   cmAnodeMainPnP1AxisZ.commandConfiguration.gearInVelocity.positionControlled := FALSE;
   cmAnodeMainPnP1AxisZ.commandConfiguration.camIn.masterOffset := 0.0;
   cmAnodeMainPnP1AxisZ.commandConfiguration.camIn.slaveOffset := 0.0;
   cmAnodeMainPnP1AxisZ.commandConfiguration.camIn.masterScaling := 1.0;
   cmAnodeMainPnP1AxisZ.commandConfiguration.camIn.slaveScaling := 1.0;
   cmAnodeMainPnP1AxisZ.commandConfiguration.camIn.masterSyncPosition := 0.0;
   cmAnodeMainPnP1AxisZ.commandConfiguration.camIn.syncProfileReference := 1;
   cmAnodeMainPnP1AxisZ.commandConfiguration.camIn.masterStartDistance := 0.0;
   cmAnodeMainPnP1AxisZ.commandConfiguration.camIn.velocity := -1.0;
   cmAnodeMainPnP1AxisZ.commandConfiguration.camIn.acceleration := -1.0;
   cmAnodeMainPnP1AxisZ.commandConfiguration.camIn.deceleration := -1.0;
   cmAnodeMainPnP1AxisZ.commandConfiguration.camIn.jerk := -1.0;
   cmAnodeMainPnP1AxisZ.commandConfiguration.camIn.applicationMode := 0;
   cmAnodeMainPnP1AxisZ.commandConfiguration.camIn.syncDirection := 1;
   cmAnodeMainPnP1AxisZ.commandConfiguration.gearOutCamOut.slavePosition := 0.0;
   cmAnodeMainPnP1AxisZ.commandConfiguration.gearOutCamOut.syncProfileReference := 1;
   cmAnodeMainPnP1AxisZ.commandConfiguration.gearOutCamOut.masterStopDistance := 0.0;
   cmAnodeMainPnP1AxisZ.commandConfiguration.gearOutCamOut.deceleration := -1.0;
   cmAnodeMainPnP1AxisZ.commandConfiguration.gearOutCamOut.jerk := -1.0;
   cmAnodeMainPnP1AxisZ.commandConfiguration.gearOutCamOut.syncOutDirection := 3;
   cmAnodeMainPnP1AxisZ.commandConfiguration.gearOutCamOut.gearOutCamOutMode := -1;
   cmAnodeMainPnP1AxisZ.commandConfiguration.phasing.phaseShift := 0.0;
   cmAnodeMainPnP1AxisZ.commandConfiguration.phasing.velocity := -1.0;
   cmAnodeMainPnP1AxisZ.commandConfiguration.phasing.acceleration := -1.0;
   cmAnodeMainPnP1AxisZ.commandConfiguration.phasing.deceleration := -1.0;
   cmAnodeMainPnP1AxisZ.commandConfiguration.phasing.jerk := -1.0;
   cmAnodeMainPnP1AxisZ.commandConfiguration.phasing.profileReference := 0;
   cmAnodeMainPnP1AxisZ.commandConfiguration.phasing.phasingDistance := 0.0;
   cmAnodeMainPnP1AxisZ.commandConfiguration.phasing.startPosition := 0.0;
   cmAnodeMainPnP1AxisZ.commandConfiguration.phasing.direction := 3;
   cmAnodeMainPnP1AxisZ.commandConfiguration.phasing.phaseAbsolute := TRUE;
   cmAnodeMainPnP1AxisZ.commandConfiguration.phasing.phaseShiftChangeOnTheFly := FALSE;
   cmAnodeMainPnP1AxisZ.commandConfiguration.offset.offset := 0.0;
   cmAnodeMainPnP1AxisZ.commandConfiguration.offset.profileReference := 1;
   cmAnodeMainPnP1AxisZ.commandConfiguration.offset.offsetDistance := 0.0;
   cmAnodeMainPnP1AxisZ.commandConfiguration.offset.startPosition := 0.0;
   cmAnodeMainPnP1AxisZ.commandConfiguration.offset.direction := 3;
   cmAnodeMainPnP1AxisZ.commandConfiguration.offset.offsetAbsolute := TRUE;
   cmAnodeMainPnP1AxisZ.commandConfiguration.offset.offsetChangeOnTheFly := FALSE;
   cmAnodeMainPnP1AxisZ.commands.enableMasterControl := TRUE;
   cmAnodeMainPnP1AxisZ.commands.enableAxis := FALSE;
   cmAnodeMainPnP1AxisZ.commands.resetAxis := FALSE;
   cmAnodeMainPnP1AxisZ.commands.openBrake := FALSE;
   cmAnodeMainPnP1AxisZ.commands.jogForward := FALSE;
   cmAnodeMainPnP1AxisZ.commands.jogBackward := FALSE;
   cmAnodeMainPnP1AxisZ.commands.moveVelocity := FALSE;
   cmAnodeMainPnP1AxisZ.commands.stop := FALSE;
   cmAnodeMainPnP1AxisZ.commands.fastStop := FALSE;
   cmAnodeMainPnP1AxisZ.commands.torqueLimiting := FALSE;
   cmAnodeMainPnP1AxisZ.commands.homing := FALSE;
   cmAnodeMainPnP1AxisZ.commands.posRelative := FALSE;
   cmAnodeMainPnP1AxisZ.commands.posAbsolute := FALSE;
   cmAnodeMainPnP1AxisZ.commands.posSuperimposed := FALSE;
   cmAnodeMainPnP1AxisZ.commands.haltSuperimposed := FALSE;
   cmAnodeMainPnP1AxisZ.commands.selectSetPosition := 3;
   cmAnodeMainPnP1AxisZ.commands.uploadParameters := FALSE;
   cmAnodeMainPnP1AxisZ.commands.refreshConfiguration := FALSE;
   cmAnodeMainPnP1AxisZ.commands.editConfiguration := FALSE;
   cmAnodeMainPnP1AxisZ.commands.saveConfiguration := FALSE;
   cmAnodeMainPnP1AxisZ.commands.uploadCurrentTorque := FALSE;
   cmAnodeMainPnP1AxisZ.commands.reset := FALSE;
   cmAnodeMainPnP1AxisZ.monitoring.enable := TRUE;
   cmAnodeMainPnP1AxisZ.monitoring.referenceDesignator := WSTRING#'AnodeMainPnP1AxisZ';
   cmAnodeMainPnP1AxisZ.monitoring.enabled := TRUE;
   cmAnodeMainPnP1AxisZ.monitoring.enableManualCmds := FALSE;
   cmAnodeMainPnP1AxisZ.monitoring.reset := FALSE;
   cmAnodeMainPnP1AxisZ.monitoring.resetAxis := FALSE;
   cmAnodeMainPnP1AxisZ.monitoring.enableAxis := TRUE;
   cmAnodeMainPnP1AxisZ.monitoring.openBrake := FALSE;
   cmAnodeMainPnP1AxisZ.monitoring.jogBackward := FALSE;
   cmAnodeMainPnP1AxisZ.monitoring.jogForward := FALSE;
   cmAnodeMainPnP1AxisZ.monitoring.moveVelocity := FALSE;
   cmAnodeMainPnP1AxisZ.monitoring.stop := FALSE;
   cmAnodeMainPnP1AxisZ.monitoring.fastStop := FALSE;
   cmAnodeMainPnP1AxisZ.monitoring.torqueLimiting := FALSE;
   cmAnodeMainPnP1AxisZ.monitoring.homing := FALSE;
   cmAnodeMainPnP1AxisZ.monitoring.posRelative := FALSE;
   cmAnodeMainPnP1AxisZ.monitoring.posAbsolute := FALSE;
   cmAnodeMainPnP1AxisZ.monitoring.posSuperimposed := FALSE;
   cmAnodeMainPnP1AxisZ.monitoring.haltSuperimposed := FALSE;
   cmAnodeMainPnP1AxisZ.monitoring.brakeOpened := FALSE;
   cmAnodeMainPnP1AxisZ.monitoring.axisEnabled := TRUE;
   cmAnodeMainPnP1AxisZ.monitoring.resetActive := FALSE;
   cmAnodeMainPnP1AxisZ.monitoring.inVelocity := FALSE;
   cmAnodeMainPnP1AxisZ.monitoring.inLimitation := FALSE;
   cmAnodeMainPnP1AxisZ.monitoring.inClamping := FALSE;
   cmAnodeMainPnP1AxisZ.monitoring.startSync := FALSE;
   cmAnodeMainPnP1AxisZ.monitoring.inSync := FALSE;
   cmAnodeMainPnP1AxisZ.monitoring.inSimulation := FALSE;
   cmAnodeMainPnP1AxisZ.monitoring.jogSelected := FALSE;
   cmAnodeMainPnP1AxisZ.monitoring.moveVelocitySelected := FALSE;
   cmAnodeMainPnP1AxisZ.monitoring.stopSelected := FALSE;
   cmAnodeMainPnP1AxisZ.monitoring.fastStopSelected := FALSE;
   cmAnodeMainPnP1AxisZ.monitoring.torqueLimitingSelected := FALSE;
   cmAnodeMainPnP1AxisZ.monitoring.homingSelected := FALSE;
   cmAnodeMainPnP1AxisZ.monitoring.posRelativeSelected := FALSE;
   cmAnodeMainPnP1AxisZ.monitoring.posAbsoluteSelected := FALSE;
   cmAnodeMainPnP1AxisZ.monitoring.posSuperimposedSelected := FALSE;
   cmAnodeMainPnP1AxisZ.monitoring.haltSuperimposedSelected := FALSE;
   cmAnodeMainPnP1AxisZ.monitoring.commandBusy := FALSE;
   cmAnodeMainPnP1AxisZ.monitoring.commandDone := FALSE;
   cmAnodeMainPnP1AxisZ.monitoring.commandAborted := FALSE;
   cmAnodeMainPnP1AxisZ.monitoring.homingCommandBusy := FALSE;
   cmAnodeMainPnP1AxisZ.monitoring.homingCommandDone := FALSE;
   cmAnodeMainPnP1AxisZ.monitoring.homingCommandAborted := FALSE;
   cmAnodeMainPnP1AxisZ.monitoring.superimposedBusy := FALSE;
   cmAnodeMainPnP1AxisZ.monitoring.superimposedDone := FALSE;
   cmAnodeMainPnP1AxisZ.monitoring.superimposedAborted := FALSE;
   cmAnodeMainPnP1AxisZ.monitoring.selectSetPosition := 3;
   cmAnodeMainPnP1AxisZ.monitoring.selectionController := FALSE;
   cmAnodeMainPnP1AxisZ.monitoring.interlockGeneral := TRUE;
   cmAnodeMainPnP1AxisZ.monitoring.interlockJogForward := TRUE;
   cmAnodeMainPnP1AxisZ.monitoring.interlockJogBackward := TRUE;
   cmAnodeMainPnP1AxisZ.monitoring.interlockWarningGeneral := FALSE;
   cmAnodeMainPnP1AxisZ.monitoring.interlockWarningJogForward := FALSE;
   cmAnodeMainPnP1AxisZ.monitoring.interlockWarningJogBackward := FALSE;
   cmAnodeMainPnP1AxisZ.monitoring.valid := TRUE;
   cmAnodeMainPnP1AxisZ.monitoring.busy := TRUE;
   cmAnodeMainPnP1AxisZ.monitoring.error := FALSE;
   cmAnodeMainPnP1AxisZ.monitoring.status := 16#7002;
   cmAnodeMainPnP1AxisZ.monitoring.subfunctionStatus := 16#0000;
   cmAnodeMainPnP1AxisZ.monitoring.actualPosition := 30.0;
   cmAnodeMainPnP1AxisZ.monitoring.actualSpeed := 0.0;
   cmAnodeMainPnP1AxisZ.monitoring.speedUnit := 1062;
   cmAnodeMainPnP1AxisZ.monitoring.positionUnit := 1013;
   cmAnodeMainPnP1AxisZ.monitoring.axisStatus1 := 16#0240_1021;
   cmAnodeMainPnP1AxisZ.monitoring.axisStatus2 := 16#0000_0000;
   cmAnodeMainPnP1AxisZ.monitoring.axisType := 1;
   cmAnodeMainPnP1AxisZ.monitoring.maxVelocity := 2500.0;
   cmAnodeMainPnP1AxisZ.monitoring.actualCurrent := 0.0;
   cmAnodeMainPnP1AxisZ.monitoring.actualTorque := 0.0;
   cmAnodeMainPnP1AxisZ.monitoring.velocityOverrideEnabled := FALSE;
   cmAnodeMainPnP1AxisZ.monitoring.sinaParaError := FALSE;
   cmAnodeMainPnP1AxisZ.monitoring.sinaParaStatus := 16#0000_0000;
   cmAnodeMainPnP1AxisZ.configuration.referenceDesignator := WSTRING#'AnodeMainPnP1AxisZ';
   cmAnodeMainPnP1AxisZ.configuration.disableAlarms := FALSE;
   cmAnodeMainPnP1AxisZ.configuration.masterControlPopUp := TRUE;
   cmAnodeMainPnP1AxisZ.configuration.setPositions[0].position := 0.0;
   cmAnodeMainPnP1AxisZ.configuration.setPositions[1..2].position := 30.0;
   cmAnodeMainPnP1AxisZ.configuration.setPositions[3..15].position := 0.0;
   cmAnodeMainPnP1AxisZ.configuration.setPositions[0..3].velocity := 50.0;
   cmAnodeMainPnP1AxisZ.configuration.setPositions[4..15].velocity := -1.0;
   cmAnodeMainPnP1AxisZ.configuration.setPositions[0..3].acceleration := 500.0;
   cmAnodeMainPnP1AxisZ.configuration.setPositions[4..15].acceleration := -1.0;
   cmAnodeMainPnP1AxisZ.configuration.setPositions[0..3].deceleration := 500.0;
   cmAnodeMainPnP1AxisZ.configuration.setPositions[4..15].deceleration := -1.0;
   cmAnodeMainPnP1AxisZ.configuration.setPositions[0..15]."name" := '';
   cmAnodeMainPnP2AxisZ.commandConfiguration.generalSettings.stopOnError := TRUE;
   cmAnodeMainPnP2AxisZ.commandConfiguration.generalSettings.resetWithRestart := FALSE;
   cmAnodeMainPnP2AxisZ.commandConfiguration.generalSettings.abortWaitingSyncCmd := TRUE;
   cmAnodeMainPnP2AxisZ.commandConfiguration.power.startMode := 1;
   cmAnodeMainPnP2AxisZ.commandConfiguration.power.stopMode := 0;
   cmAnodeMainPnP2AxisZ.commandConfiguration.power.syncMotionSimulation := FALSE;
   cmAnodeMainPnP2AxisZ.commandConfiguration.power.syncMotionSimulationExtendedMode := -1;
   cmAnodeMainPnP2AxisZ.commandConfiguration.jog.velocity := 10.0;
   cmAnodeMainPnP2AxisZ.commandConfiguration.jog.acceleration := 100.0;
   cmAnodeMainPnP2AxisZ.commandConfiguration.jog.deceleration := 100.0;
   cmAnodeMainPnP2AxisZ.commandConfiguration.jog.jerk := -1.0;
   cmAnodeMainPnP2AxisZ.commandConfiguration.jog.positionControlled := TRUE;
   cmAnodeMainPnP2AxisZ.commandConfiguration.jog.increment := 0.0;
   cmAnodeMainPnP2AxisZ.commandConfiguration.jog.mode := 0;
   cmAnodeMainPnP2AxisZ.commandConfiguration.moveVelocity.velocity := 10.0;
   cmAnodeMainPnP2AxisZ.commandConfiguration.moveVelocity.acceleration := 100.0;
   cmAnodeMainPnP2AxisZ.commandConfiguration.moveVelocity.deceleration := 100.0;
   cmAnodeMainPnP2AxisZ.commandConfiguration.moveVelocity.jerk := -1.0;
   cmAnodeMainPnP2AxisZ.commandConfiguration.moveVelocity.direction := 0;
   cmAnodeMainPnP2AxisZ.commandConfiguration.moveVelocity.positionControlled := TRUE;
   cmAnodeMainPnP2AxisZ.commandConfiguration.moveVelocity.velocityChangeOnTheFly := FALSE;
   cmAnodeMainPnP2AxisZ.commandConfiguration.stop.deceleration := -1.0;
   cmAnodeMainPnP2AxisZ.commandConfiguration.stop.jerk := -1.0;
   cmAnodeMainPnP2AxisZ.commandConfiguration.stop.abortAcceleration := FALSE;
   cmAnodeMainPnP2AxisZ.commandConfiguration.fastStop.deceleration := -1.0;
   cmAnodeMainPnP2AxisZ.commandConfiguration.fastStop.jerk := -1.0;
   cmAnodeMainPnP2AxisZ.commandConfiguration.fastStop.abortAcceleration := FALSE;
   cmAnodeMainPnP2AxisZ.commandConfiguration.fastStop.replaceStopPossible := FALSE;
   cmAnodeMainPnP2AxisZ.commandConfiguration.torqueLimiting.limit := -1.0;
   cmAnodeMainPnP2AxisZ.commandConfiguration.torqueLimiting.mode := 0;
   cmAnodeMainPnP2AxisZ.commandConfiguration.homing.position := 0.0;
   cmAnodeMainPnP2AxisZ.commandConfiguration.homing.mode := 0;
   cmAnodeMainPnP2AxisZ.commandConfiguration.homing.sensor := 0;
   cmAnodeMainPnP2AxisZ.commandConfiguration.homing.extendedMode := -1;
   cmAnodeMainPnP2AxisZ.commandConfiguration.homing.extendedModeTorqueLimit := 0.0;
   cmAnodeMainPnP2AxisZ.commandConfiguration.homing.extendedModeTargetPosition := 0.0;
   cmAnodeMainPnP2AxisZ.commandConfiguration.posRelative.distance := 0.0;
   cmAnodeMainPnP2AxisZ.commandConfiguration.posRelative.velocity := 10.0;
   cmAnodeMainPnP2AxisZ.commandConfiguration.posRelative.acceleration := 100.0;
   cmAnodeMainPnP2AxisZ.commandConfiguration.posRelative.deceleration := 100.0;
   cmAnodeMainPnP2AxisZ.commandConfiguration.posRelative.jerk := -1.0;
   cmAnodeMainPnP2AxisZ.commandConfiguration.posRelative.direction := 0;
   cmAnodeMainPnP2AxisZ.commandConfiguration.posAbsolute.position := 0.0;
   cmAnodeMainPnP2AxisZ.commandConfiguration.posAbsolute.velocity := -1.0;
   cmAnodeMainPnP2AxisZ.commandConfiguration.posAbsolute.acceleration := -1.0;
   cmAnodeMainPnP2AxisZ.commandConfiguration.posAbsolute.deceleration := -1.0;
   cmAnodeMainPnP2AxisZ.commandConfiguration.posAbsolute.jerk := -1.0;
   cmAnodeMainPnP2AxisZ.commandConfiguration.posAbsolute.direction := 1;
   cmAnodeMainPnP2AxisZ.commandConfiguration.posAbsolute.positionChangeOnTheFly := FALSE;
   cmAnodeMainPnP2AxisZ.commandConfiguration.posAbsolute.velocityChangeOnTheFly := FALSE;
   cmAnodeMainPnP2AxisZ.commandConfiguration.posSuperimposed.distance := 0.0;
   cmAnodeMainPnP2AxisZ.commandConfiguration.posSuperimposed.velocityDiff := -1.0;
   cmAnodeMainPnP2AxisZ.commandConfiguration.posSuperimposed.acceleration := -1.0;
   cmAnodeMainPnP2AxisZ.commandConfiguration.posSuperimposed.deceleration := -1.0;
   cmAnodeMainPnP2AxisZ.commandConfiguration.posSuperimposed.jerk := -1.0;
   cmAnodeMainPnP2AxisZ.commandConfiguration.posSuperimposed.direction := 0;
   cmAnodeMainPnP2AxisZ.commandConfiguration.haltSuperimposed.deceleration := -1.0;
   cmAnodeMainPnP2AxisZ.commandConfiguration.haltSuperimposed.jerk := -1.0;
   cmAnodeMainPnP2AxisZ.commandConfiguration.haltSuperimposed.abortAcceleration := FALSE;
   cmAnodeMainPnP2AxisZ.commandConfiguration.gearInRelative.ratioNumerator := 1;
   cmAnodeMainPnP2AxisZ.commandConfiguration.gearInRelative.ratioDenominator := 1;
   cmAnodeMainPnP2AxisZ.commandConfiguration.gearInRelative.acceleration := -1.0;
   cmAnodeMainPnP2AxisZ.commandConfiguration.gearInRelative.deceleration := -1.0;
   cmAnodeMainPnP2AxisZ.commandConfiguration.gearInRelative.jerk := -1.0;
   cmAnodeMainPnP2AxisZ.commandConfiguration.gearInRelative.ratioChangeOnTheFly := FALSE;
   cmAnodeMainPnP2AxisZ.commandConfiguration.gearInAbsolute.ratioNumerator := 1;
   cmAnodeMainPnP2AxisZ.commandConfiguration.gearInAbsolute.ratioDenominator := 1;
   cmAnodeMainPnP2AxisZ.commandConfiguration.gearInAbsolute.masterSyncPosition := 0.0;
   cmAnodeMainPnP2AxisZ.commandConfiguration.gearInAbsolute.slaveSyncPosition := 0.0;
   cmAnodeMainPnP2AxisZ.commandConfiguration.gearInAbsolute.syncProfileReference := 1;
   cmAnodeMainPnP2AxisZ.commandConfiguration.gearInAbsolute.masterStartDistance := 0.0;
   cmAnodeMainPnP2AxisZ.commandConfiguration.gearInAbsolute.velocity := -1.0;
   cmAnodeMainPnP2AxisZ.commandConfiguration.gearInAbsolute.acceleration := -1.0;
   cmAnodeMainPnP2AxisZ.commandConfiguration.gearInAbsolute.deceleration := -1.0;
   cmAnodeMainPnP2AxisZ.commandConfiguration.gearInAbsolute.jerk := -1.0;
   cmAnodeMainPnP2AxisZ.commandConfiguration.gearInAbsolute.syncDirection := 1;
   cmAnodeMainPnP2AxisZ.commandConfiguration.gearInAbsolute.ratioChangeOnTheFly := FALSE;
   cmAnodeMainPnP2AxisZ.commandConfiguration.gearInVelocity.continuousUpdate := FALSE;
   cmAnodeMainPnP2AxisZ.commandConfiguration.gearInVelocity.ratioNumerator := 1;
   cmAnodeMainPnP2AxisZ.commandConfiguration.gearInVelocity.ratioDenominator := 1;
   cmAnodeMainPnP2AxisZ.commandConfiguration.gearInVelocity.acceleration := -1.0;
   cmAnodeMainPnP2AxisZ.commandConfiguration.gearInVelocity.deceleration := -1.0;
   cmAnodeMainPnP2AxisZ.commandConfiguration.gearInVelocity.jerk := -1.0;
   cmAnodeMainPnP2AxisZ.commandConfiguration.gearInVelocity.positionControlled := FALSE;
   cmAnodeMainPnP2AxisZ.commandConfiguration.camIn.masterOffset := 0.0;
   cmAnodeMainPnP2AxisZ.commandConfiguration.camIn.slaveOffset := 0.0;
   cmAnodeMainPnP2AxisZ.commandConfiguration.camIn.masterScaling := 1.0;
   cmAnodeMainPnP2AxisZ.commandConfiguration.camIn.slaveScaling := 1.0;
   cmAnodeMainPnP2AxisZ.commandConfiguration.camIn.masterSyncPosition := 0.0;
   cmAnodeMainPnP2AxisZ.commandConfiguration.camIn.syncProfileReference := 1;
   cmAnodeMainPnP2AxisZ.commandConfiguration.camIn.masterStartDistance := 0.0;
   cmAnodeMainPnP2AxisZ.commandConfiguration.camIn.velocity := -1.0;
   cmAnodeMainPnP2AxisZ.commandConfiguration.camIn.acceleration := -1.0;
   cmAnodeMainPnP2AxisZ.commandConfiguration.camIn.deceleration := -1.0;
   cmAnodeMainPnP2AxisZ.commandConfiguration.camIn.jerk := -1.0;
   cmAnodeMainPnP2AxisZ.commandConfiguration.camIn.applicationMode := 0;
   cmAnodeMainPnP2AxisZ.commandConfiguration.camIn.syncDirection := 1;
   cmAnodeMainPnP2AxisZ.commandConfiguration.gearOutCamOut.slavePosition := 0.0;
   cmAnodeMainPnP2AxisZ.commandConfiguration.gearOutCamOut.syncProfileReference := 1;
   cmAnodeMainPnP2AxisZ.commandConfiguration.gearOutCamOut.masterStopDistance := 0.0;
   cmAnodeMainPnP2AxisZ.commandConfiguration.gearOutCamOut.deceleration := -1.0;
   cmAnodeMainPnP2AxisZ.commandConfiguration.gearOutCamOut.jerk := -1.0;
   cmAnodeMainPnP2AxisZ.commandConfiguration.gearOutCamOut.syncOutDirection := 3;
   cmAnodeMainPnP2AxisZ.commandConfiguration.gearOutCamOut.gearOutCamOutMode := -1;
   cmAnodeMainPnP2AxisZ.commandConfiguration.phasing.phaseShift := 0.0;
   cmAnodeMainPnP2AxisZ.commandConfiguration.phasing.velocity := -1.0;
   cmAnodeMainPnP2AxisZ.commandConfiguration.phasing.acceleration := -1.0;
   cmAnodeMainPnP2AxisZ.commandConfiguration.phasing.deceleration := -1.0;
   cmAnodeMainPnP2AxisZ.commandConfiguration.phasing.jerk := -1.0;
   cmAnodeMainPnP2AxisZ.commandConfiguration.phasing.profileReference := 0;
   cmAnodeMainPnP2AxisZ.commandConfiguration.phasing.phasingDistance := 0.0;
   cmAnodeMainPnP2AxisZ.commandConfiguration.phasing.startPosition := 0.0;
   cmAnodeMainPnP2AxisZ.commandConfiguration.phasing.direction := 3;
   cmAnodeMainPnP2AxisZ.commandConfiguration.phasing.phaseAbsolute := TRUE;
   cmAnodeMainPnP2AxisZ.commandConfiguration.phasing.phaseShiftChangeOnTheFly := FALSE;
   cmAnodeMainPnP2AxisZ.commandConfiguration.offset.offset := 0.0;
   cmAnodeMainPnP2AxisZ.commandConfiguration.offset.profileReference := 1;
   cmAnodeMainPnP2AxisZ.commandConfiguration.offset.offsetDistance := 0.0;
   cmAnodeMainPnP2AxisZ.commandConfiguration.offset.startPosition := 0.0;
   cmAnodeMainPnP2AxisZ.commandConfiguration.offset.direction := 3;
   cmAnodeMainPnP2AxisZ.commandConfiguration.offset.offsetAbsolute := TRUE;
   cmAnodeMainPnP2AxisZ.commandConfiguration.offset.offsetChangeOnTheFly := FALSE;
   cmAnodeMainPnP2AxisZ.commands.enableMasterControl := TRUE;
   cmAnodeMainPnP2AxisZ.commands.enableAxis := FALSE;
   cmAnodeMainPnP2AxisZ.commands.resetAxis := FALSE;
   cmAnodeMainPnP2AxisZ.commands.openBrake := FALSE;
   cmAnodeMainPnP2AxisZ.commands.jogForward := FALSE;
   cmAnodeMainPnP2AxisZ.commands.jogBackward := FALSE;
   cmAnodeMainPnP2AxisZ.commands.moveVelocity := FALSE;
   cmAnodeMainPnP2AxisZ.commands.stop := FALSE;
   cmAnodeMainPnP2AxisZ.commands.fastStop := FALSE;
   cmAnodeMainPnP2AxisZ.commands.torqueLimiting := FALSE;
   cmAnodeMainPnP2AxisZ.commands.homing := FALSE;
   cmAnodeMainPnP2AxisZ.commands.posRelative := FALSE;
   cmAnodeMainPnP2AxisZ.commands.posAbsolute := FALSE;
   cmAnodeMainPnP2AxisZ.commands.posSuperimposed := FALSE;
   cmAnodeMainPnP2AxisZ.commands.haltSuperimposed := FALSE;
   cmAnodeMainPnP2AxisZ.commands.selectSetPosition := 3;
   cmAnodeMainPnP2AxisZ.commands.uploadParameters := FALSE;
   cmAnodeMainPnP2AxisZ.commands.refreshConfiguration := FALSE;
   cmAnodeMainPnP2AxisZ.commands.editConfiguration := FALSE;
   cmAnodeMainPnP2AxisZ.commands.saveConfiguration := FALSE;
   cmAnodeMainPnP2AxisZ.commands.uploadCurrentTorque := FALSE;
   cmAnodeMainPnP2AxisZ.commands.reset := FALSE;
   cmAnodeMainPnP2AxisZ.monitoring.enable := TRUE;
   cmAnodeMainPnP2AxisZ.monitoring.referenceDesignator := WSTRING#'AnodeMainPnP2AxisZ';
   cmAnodeMainPnP2AxisZ.monitoring.enabled := TRUE;
   cmAnodeMainPnP2AxisZ.monitoring.enableManualCmds := FALSE;
   cmAnodeMainPnP2AxisZ.monitoring.reset := FALSE;
   cmAnodeMainPnP2AxisZ.monitoring.resetAxis := FALSE;
   cmAnodeMainPnP2AxisZ.monitoring.enableAxis := TRUE;
   cmAnodeMainPnP2AxisZ.monitoring.openBrake := FALSE;
   cmAnodeMainPnP2AxisZ.monitoring.jogBackward := FALSE;
   cmAnodeMainPnP2AxisZ.monitoring.jogForward := FALSE;
   cmAnodeMainPnP2AxisZ.monitoring.moveVelocity := FALSE;
   cmAnodeMainPnP2AxisZ.monitoring.stop := FALSE;
   cmAnodeMainPnP2AxisZ.monitoring.fastStop := FALSE;
   cmAnodeMainPnP2AxisZ.monitoring.torqueLimiting := FALSE;
   cmAnodeMainPnP2AxisZ.monitoring.homing := FALSE;
   cmAnodeMainPnP2AxisZ.monitoring.posRelative := FALSE;
   cmAnodeMainPnP2AxisZ.monitoring.posAbsolute := FALSE;
   cmAnodeMainPnP2AxisZ.monitoring.posSuperimposed := FALSE;
   cmAnodeMainPnP2AxisZ.monitoring.haltSuperimposed := FALSE;
   cmAnodeMainPnP2AxisZ.monitoring.brakeOpened := FALSE;
   cmAnodeMainPnP2AxisZ.monitoring.axisEnabled := TRUE;
   cmAnodeMainPnP2AxisZ.monitoring.resetActive := FALSE;
   cmAnodeMainPnP2AxisZ.monitoring.inVelocity := FALSE;
   cmAnodeMainPnP2AxisZ.monitoring.inLimitation := FALSE;
   cmAnodeMainPnP2AxisZ.monitoring.inClamping := FALSE;
   cmAnodeMainPnP2AxisZ.monitoring.startSync := FALSE;
   cmAnodeMainPnP2AxisZ.monitoring.inSync := FALSE;
   cmAnodeMainPnP2AxisZ.monitoring.inSimulation := FALSE;
   cmAnodeMainPnP2AxisZ.monitoring.jogSelected := FALSE;
   cmAnodeMainPnP2AxisZ.monitoring.moveVelocitySelected := FALSE;
   cmAnodeMainPnP2AxisZ.monitoring.stopSelected := FALSE;
   cmAnodeMainPnP2AxisZ.monitoring.fastStopSelected := FALSE;
   cmAnodeMainPnP2AxisZ.monitoring.torqueLimitingSelected := FALSE;
   cmAnodeMainPnP2AxisZ.monitoring.homingSelected := FALSE;
   cmAnodeMainPnP2AxisZ.monitoring.posRelativeSelected := FALSE;
   cmAnodeMainPnP2AxisZ.monitoring.posAbsoluteSelected := FALSE;
   cmAnodeMainPnP2AxisZ.monitoring.posSuperimposedSelected := FALSE;
   cmAnodeMainPnP2AxisZ.monitoring.haltSuperimposedSelected := FALSE;
   cmAnodeMainPnP2AxisZ.monitoring.commandBusy := FALSE;
   cmAnodeMainPnP2AxisZ.monitoring.commandDone := FALSE;
   cmAnodeMainPnP2AxisZ.monitoring.commandAborted := FALSE;
   cmAnodeMainPnP2AxisZ.monitoring.homingCommandBusy := FALSE;
   cmAnodeMainPnP2AxisZ.monitoring.homingCommandDone := FALSE;
   cmAnodeMainPnP2AxisZ.monitoring.homingCommandAborted := FALSE;
   cmAnodeMainPnP2AxisZ.monitoring.superimposedBusy := FALSE;
   cmAnodeMainPnP2AxisZ.monitoring.superimposedDone := FALSE;
   cmAnodeMainPnP2AxisZ.monitoring.superimposedAborted := FALSE;
   cmAnodeMainPnP2AxisZ.monitoring.selectSetPosition := 3;
   cmAnodeMainPnP2AxisZ.monitoring.selectionController := FALSE;
   cmAnodeMainPnP2AxisZ.monitoring.interlockGeneral := TRUE;
   cmAnodeMainPnP2AxisZ.monitoring.interlockJogForward := TRUE;
   cmAnodeMainPnP2AxisZ.monitoring.interlockJogBackward := TRUE;
   cmAnodeMainPnP2AxisZ.monitoring.interlockWarningGeneral := FALSE;
   cmAnodeMainPnP2AxisZ.monitoring.interlockWarningJogForward := FALSE;
   cmAnodeMainPnP2AxisZ.monitoring.interlockWarningJogBackward := FALSE;
   cmAnodeMainPnP2AxisZ.monitoring.valid := TRUE;
   cmAnodeMainPnP2AxisZ.monitoring.busy := TRUE;
   cmAnodeMainPnP2AxisZ.monitoring.error := FALSE;
   cmAnodeMainPnP2AxisZ.monitoring.status := 16#7002;
   cmAnodeMainPnP2AxisZ.monitoring.subfunctionStatus := 16#0000;
   cmAnodeMainPnP2AxisZ.monitoring.actualPosition := 30.0;
   cmAnodeMainPnP2AxisZ.monitoring.actualSpeed := 0.0;
   cmAnodeMainPnP2AxisZ.monitoring.speedUnit := 1062;
   cmAnodeMainPnP2AxisZ.monitoring.positionUnit := 1013;
   cmAnodeMainPnP2AxisZ.monitoring.axisStatus1 := 16#0240_1021;
   cmAnodeMainPnP2AxisZ.monitoring.axisStatus2 := 16#0000_0000;
   cmAnodeMainPnP2AxisZ.monitoring.axisType := 1;
   cmAnodeMainPnP2AxisZ.monitoring.maxVelocity := 2500.0;
   cmAnodeMainPnP2AxisZ.monitoring.actualCurrent := 0.0;
   cmAnodeMainPnP2AxisZ.monitoring.actualTorque := 0.0;
   cmAnodeMainPnP2AxisZ.monitoring.velocityOverrideEnabled := FALSE;
   cmAnodeMainPnP2AxisZ.monitoring.sinaParaError := FALSE;
   cmAnodeMainPnP2AxisZ.monitoring.sinaParaStatus := 16#0000_0000;
   cmAnodeMainPnP2AxisZ.configuration.referenceDesignator := WSTRING#'AnodeMainPnP2AxisZ';
   cmAnodeMainPnP2AxisZ.configuration.disableAlarms := FALSE;
   cmAnodeMainPnP2AxisZ.configuration.masterControlPopUp := TRUE;
   cmAnodeMainPnP2AxisZ.configuration.setPositions[0].position := 0.0;
   cmAnodeMainPnP2AxisZ.configuration.setPositions[1..2].position := 30.0;
   cmAnodeMainPnP2AxisZ.configuration.setPositions[3..15].position := 0.0;
   cmAnodeMainPnP2AxisZ.configuration.setPositions[0..3].velocity := 50.0;
   cmAnodeMainPnP2AxisZ.configuration.setPositions[4..15].velocity := -1.0;
   cmAnodeMainPnP2AxisZ.configuration.setPositions[0..3].acceleration := 500.0;
   cmAnodeMainPnP2AxisZ.configuration.setPositions[4..15].acceleration := -1.0;
   cmAnodeMainPnP2AxisZ.configuration.setPositions[0..3].deceleration := 500.0;
   cmAnodeMainPnP2AxisZ.configuration.setPositions[4..15].deceleration := -1.0;
   cmAnodeMainPnP2AxisZ.configuration.setPositions[0..15]."name" := '';
   cmAnodeAlignTableAxisX.commandConfiguration.generalSettings.stopOnError := TRUE;
   cmAnodeAlignTableAxisX.commandConfiguration.generalSettings.resetWithRestart := FALSE;
   cmAnodeAlignTableAxisX.commandConfiguration.generalSettings.abortWaitingSyncCmd := TRUE;
   cmAnodeAlignTableAxisX.commandConfiguration.power.startMode := 1;
   cmAnodeAlignTableAxisX.commandConfiguration.power.stopMode := 0;
   cmAnodeAlignTableAxisX.commandConfiguration.power.syncMotionSimulation := FALSE;
   cmAnodeAlignTableAxisX.commandConfiguration.power.syncMotionSimulationExtendedMode := -1;
   cmAnodeAlignTableAxisX.commandConfiguration.jog.velocity := 10.0;
   cmAnodeAlignTableAxisX.commandConfiguration.jog.acceleration := 100.0;
   cmAnodeAlignTableAxisX.commandConfiguration.jog.deceleration := 100.0;
   cmAnodeAlignTableAxisX.commandConfiguration.jog.jerk := -1.0;
   cmAnodeAlignTableAxisX.commandConfiguration.jog.positionControlled := TRUE;
   cmAnodeAlignTableAxisX.commandConfiguration.jog.increment := 0.0;
   cmAnodeAlignTableAxisX.commandConfiguration.jog.mode := 0;
   cmAnodeAlignTableAxisX.commandConfiguration.moveVelocity.velocity := 10.0;
   cmAnodeAlignTableAxisX.commandConfiguration.moveVelocity.acceleration := 100.0;
   cmAnodeAlignTableAxisX.commandConfiguration.moveVelocity.deceleration := 100.0;
   cmAnodeAlignTableAxisX.commandConfiguration.moveVelocity.jerk := -1.0;
   cmAnodeAlignTableAxisX.commandConfiguration.moveVelocity.direction := 0;
   cmAnodeAlignTableAxisX.commandConfiguration.moveVelocity.positionControlled := TRUE;
   cmAnodeAlignTableAxisX.commandConfiguration.moveVelocity.velocityChangeOnTheFly := FALSE;
   cmAnodeAlignTableAxisX.commandConfiguration.stop.deceleration := -1.0;
   cmAnodeAlignTableAxisX.commandConfiguration.stop.jerk := -1.0;
   cmAnodeAlignTableAxisX.commandConfiguration.stop.abortAcceleration := FALSE;
   cmAnodeAlignTableAxisX.commandConfiguration.fastStop.deceleration := -1.0;
   cmAnodeAlignTableAxisX.commandConfiguration.fastStop.jerk := -1.0;
   cmAnodeAlignTableAxisX.commandConfiguration.fastStop.abortAcceleration := FALSE;
   cmAnodeAlignTableAxisX.commandConfiguration.fastStop.replaceStopPossible := FALSE;
   cmAnodeAlignTableAxisX.commandConfiguration.torqueLimiting.limit := -1.0;
   cmAnodeAlignTableAxisX.commandConfiguration.torqueLimiting.mode := 0;
   cmAnodeAlignTableAxisX.commandConfiguration.homing.position := 0.0;
   cmAnodeAlignTableAxisX.commandConfiguration.homing.mode := 0;
   cmAnodeAlignTableAxisX.commandConfiguration.homing.sensor := 0;
   cmAnodeAlignTableAxisX.commandConfiguration.homing.extendedMode := -1;
   cmAnodeAlignTableAxisX.commandConfiguration.homing.extendedModeTorqueLimit := 0.0;
   cmAnodeAlignTableAxisX.commandConfiguration.homing.extendedModeTargetPosition := 0.0;
   cmAnodeAlignTableAxisX.commandConfiguration.posRelative.distance := 0.0;
   cmAnodeAlignTableAxisX.commandConfiguration.posRelative.velocity := 10.0;
   cmAnodeAlignTableAxisX.commandConfiguration.posRelative.acceleration := 100.0;
   cmAnodeAlignTableAxisX.commandConfiguration.posRelative.deceleration := 100.0;
   cmAnodeAlignTableAxisX.commandConfiguration.posRelative.jerk := -1.0;
   cmAnodeAlignTableAxisX.commandConfiguration.posRelative.direction := 0;
   cmAnodeAlignTableAxisX.commandConfiguration.posAbsolute.position := 0.0;
   cmAnodeAlignTableAxisX.commandConfiguration.posAbsolute.velocity := -1.0;
   cmAnodeAlignTableAxisX.commandConfiguration.posAbsolute.acceleration := -1.0;
   cmAnodeAlignTableAxisX.commandConfiguration.posAbsolute.deceleration := -1.0;
   cmAnodeAlignTableAxisX.commandConfiguration.posAbsolute.jerk := -1.0;
   cmAnodeAlignTableAxisX.commandConfiguration.posAbsolute.direction := 1;
   cmAnodeAlignTableAxisX.commandConfiguration.posAbsolute.positionChangeOnTheFly := FALSE;
   cmAnodeAlignTableAxisX.commandConfiguration.posAbsolute.velocityChangeOnTheFly := FALSE;
   cmAnodeAlignTableAxisX.commandConfiguration.posSuperimposed.distance := 0.0;
   cmAnodeAlignTableAxisX.commandConfiguration.posSuperimposed.velocityDiff := -1.0;
   cmAnodeAlignTableAxisX.commandConfiguration.posSuperimposed.acceleration := -1.0;
   cmAnodeAlignTableAxisX.commandConfiguration.posSuperimposed.deceleration := -1.0;
   cmAnodeAlignTableAxisX.commandConfiguration.posSuperimposed.jerk := -1.0;
   cmAnodeAlignTableAxisX.commandConfiguration.posSuperimposed.direction := 0;
   cmAnodeAlignTableAxisX.commandConfiguration.haltSuperimposed.deceleration := -1.0;
   cmAnodeAlignTableAxisX.commandConfiguration.haltSuperimposed.jerk := -1.0;
   cmAnodeAlignTableAxisX.commandConfiguration.haltSuperimposed.abortAcceleration := FALSE;
   cmAnodeAlignTableAxisX.commandConfiguration.gearInRelative.ratioNumerator := 1;
   cmAnodeAlignTableAxisX.commandConfiguration.gearInRelative.ratioDenominator := 1;
   cmAnodeAlignTableAxisX.commandConfiguration.gearInRelative.acceleration := -1.0;
   cmAnodeAlignTableAxisX.commandConfiguration.gearInRelative.deceleration := -1.0;
   cmAnodeAlignTableAxisX.commandConfiguration.gearInRelative.jerk := -1.0;
   cmAnodeAlignTableAxisX.commandConfiguration.gearInRelative.ratioChangeOnTheFly := FALSE;
   cmAnodeAlignTableAxisX.commandConfiguration.gearInAbsolute.ratioNumerator := 1;
   cmAnodeAlignTableAxisX.commandConfiguration.gearInAbsolute.ratioDenominator := 1;
   cmAnodeAlignTableAxisX.commandConfiguration.gearInAbsolute.masterSyncPosition := 0.0;
   cmAnodeAlignTableAxisX.commandConfiguration.gearInAbsolute.slaveSyncPosition := 0.0;
   cmAnodeAlignTableAxisX.commandConfiguration.gearInAbsolute.syncProfileReference := 1;
   cmAnodeAlignTableAxisX.commandConfiguration.gearInAbsolute.masterStartDistance := 0.0;
   cmAnodeAlignTableAxisX.commandConfiguration.gearInAbsolute.velocity := -1.0;
   cmAnodeAlignTableAxisX.commandConfiguration.gearInAbsolute.acceleration := -1.0;
   cmAnodeAlignTableAxisX.commandConfiguration.gearInAbsolute.deceleration := -1.0;
   cmAnodeAlignTableAxisX.commandConfiguration.gearInAbsolute.jerk := -1.0;
   cmAnodeAlignTableAxisX.commandConfiguration.gearInAbsolute.syncDirection := 1;
   cmAnodeAlignTableAxisX.commandConfiguration.gearInAbsolute.ratioChangeOnTheFly := FALSE;
   cmAnodeAlignTableAxisX.commandConfiguration.gearInVelocity.continuousUpdate := FALSE;
   cmAnodeAlignTableAxisX.commandConfiguration.gearInVelocity.ratioNumerator := 1;
   cmAnodeAlignTableAxisX.commandConfiguration.gearInVelocity.ratioDenominator := 1;
   cmAnodeAlignTableAxisX.commandConfiguration.gearInVelocity.acceleration := -1.0;
   cmAnodeAlignTableAxisX.commandConfiguration.gearInVelocity.deceleration := -1.0;
   cmAnodeAlignTableAxisX.commandConfiguration.gearInVelocity.jerk := -1.0;
   cmAnodeAlignTableAxisX.commandConfiguration.gearInVelocity.positionControlled := FALSE;
   cmAnodeAlignTableAxisX.commandConfiguration.camIn.masterOffset := 0.0;
   cmAnodeAlignTableAxisX.commandConfiguration.camIn.slaveOffset := 0.0;
   cmAnodeAlignTableAxisX.commandConfiguration.camIn.masterScaling := 1.0;
   cmAnodeAlignTableAxisX.commandConfiguration.camIn.slaveScaling := 1.0;
   cmAnodeAlignTableAxisX.commandConfiguration.camIn.masterSyncPosition := 0.0;
   cmAnodeAlignTableAxisX.commandConfiguration.camIn.syncProfileReference := 1;
   cmAnodeAlignTableAxisX.commandConfiguration.camIn.masterStartDistance := 0.0;
   cmAnodeAlignTableAxisX.commandConfiguration.camIn.velocity := -1.0;
   cmAnodeAlignTableAxisX.commandConfiguration.camIn.acceleration := -1.0;
   cmAnodeAlignTableAxisX.commandConfiguration.camIn.deceleration := -1.0;
   cmAnodeAlignTableAxisX.commandConfiguration.camIn.jerk := -1.0;
   cmAnodeAlignTableAxisX.commandConfiguration.camIn.applicationMode := 0;
   cmAnodeAlignTableAxisX.commandConfiguration.camIn.syncDirection := 1;
   cmAnodeAlignTableAxisX.commandConfiguration.gearOutCamOut.slavePosition := 0.0;
   cmAnodeAlignTableAxisX.commandConfiguration.gearOutCamOut.syncProfileReference := 1;
   cmAnodeAlignTableAxisX.commandConfiguration.gearOutCamOut.masterStopDistance := 0.0;
   cmAnodeAlignTableAxisX.commandConfiguration.gearOutCamOut.deceleration := -1.0;
   cmAnodeAlignTableAxisX.commandConfiguration.gearOutCamOut.jerk := -1.0;
   cmAnodeAlignTableAxisX.commandConfiguration.gearOutCamOut.syncOutDirection := 3;
   cmAnodeAlignTableAxisX.commandConfiguration.gearOutCamOut.gearOutCamOutMode := -1;
   cmAnodeAlignTableAxisX.commandConfiguration.phasing.phaseShift := 0.0;
   cmAnodeAlignTableAxisX.commandConfiguration.phasing.velocity := -1.0;
   cmAnodeAlignTableAxisX.commandConfiguration.phasing.acceleration := -1.0;
   cmAnodeAlignTableAxisX.commandConfiguration.phasing.deceleration := -1.0;
   cmAnodeAlignTableAxisX.commandConfiguration.phasing.jerk := -1.0;
   cmAnodeAlignTableAxisX.commandConfiguration.phasing.profileReference := 0;
   cmAnodeAlignTableAxisX.commandConfiguration.phasing.phasingDistance := 0.0;
   cmAnodeAlignTableAxisX.commandConfiguration.phasing.startPosition := 0.0;
   cmAnodeAlignTableAxisX.commandConfiguration.phasing.direction := 3;
   cmAnodeAlignTableAxisX.commandConfiguration.phasing.phaseAbsolute := TRUE;
   cmAnodeAlignTableAxisX.commandConfiguration.phasing.phaseShiftChangeOnTheFly := FALSE;
   cmAnodeAlignTableAxisX.commandConfiguration.offset.offset := 0.0;
   cmAnodeAlignTableAxisX.commandConfiguration.offset.profileReference := 1;
   cmAnodeAlignTableAxisX.commandConfiguration.offset.offsetDistance := 0.0;
   cmAnodeAlignTableAxisX.commandConfiguration.offset.startPosition := 0.0;
   cmAnodeAlignTableAxisX.commandConfiguration.offset.direction := 3;
   cmAnodeAlignTableAxisX.commandConfiguration.offset.offsetAbsolute := TRUE;
   cmAnodeAlignTableAxisX.commandConfiguration.offset.offsetChangeOnTheFly := FALSE;
   cmAnodeAlignTableAxisX.commands.enableMasterControl := TRUE;
   cmAnodeAlignTableAxisX.commands.enableAxis := FALSE;
   cmAnodeAlignTableAxisX.commands.resetAxis := FALSE;
   cmAnodeAlignTableAxisX.commands.openBrake := FALSE;
   cmAnodeAlignTableAxisX.commands.jogForward := FALSE;
   cmAnodeAlignTableAxisX.commands.jogBackward := FALSE;
   cmAnodeAlignTableAxisX.commands.moveVelocity := FALSE;
   cmAnodeAlignTableAxisX.commands.stop := FALSE;
   cmAnodeAlignTableAxisX.commands.fastStop := FALSE;
   cmAnodeAlignTableAxisX.commands.torqueLimiting := FALSE;
   cmAnodeAlignTableAxisX.commands.homing := FALSE;
   cmAnodeAlignTableAxisX.commands.posRelative := FALSE;
   cmAnodeAlignTableAxisX.commands.posAbsolute := FALSE;
   cmAnodeAlignTableAxisX.commands.posSuperimposed := FALSE;
   cmAnodeAlignTableAxisX.commands.haltSuperimposed := FALSE;
   cmAnodeAlignTableAxisX.commands.selectSetPosition := -1;
   cmAnodeAlignTableAxisX.commands.uploadParameters := FALSE;
   cmAnodeAlignTableAxisX.commands.refreshConfiguration := FALSE;
   cmAnodeAlignTableAxisX.commands.editConfiguration := FALSE;
   cmAnodeAlignTableAxisX.commands.saveConfiguration := FALSE;
   cmAnodeAlignTableAxisX.commands.uploadCurrentTorque := FALSE;
   cmAnodeAlignTableAxisX.commands.reset := FALSE;
   cmAnodeAlignTableAxisX.monitoring.enable := TRUE;
   cmAnodeAlignTableAxisX.monitoring.referenceDesignator := WSTRING#'AnodeAlignTableAxisX';
   cmAnodeAlignTableAxisX.monitoring.enabled := TRUE;
   cmAnodeAlignTableAxisX.monitoring.enableManualCmds := FALSE;
   cmAnodeAlignTableAxisX.monitoring.reset := FALSE;
   cmAnodeAlignTableAxisX.monitoring.resetAxis := FALSE;
   cmAnodeAlignTableAxisX.monitoring.enableAxis := TRUE;
   cmAnodeAlignTableAxisX.monitoring.openBrake := FALSE;
   cmAnodeAlignTableAxisX.monitoring.jogBackward := FALSE;
   cmAnodeAlignTableAxisX.monitoring.jogForward := FALSE;
   cmAnodeAlignTableAxisX.monitoring.moveVelocity := FALSE;
   cmAnodeAlignTableAxisX.monitoring.stop := FALSE;
   cmAnodeAlignTableAxisX.monitoring.fastStop := FALSE;
   cmAnodeAlignTableAxisX.monitoring.torqueLimiting := FALSE;
   cmAnodeAlignTableAxisX.monitoring.homing := FALSE;
   cmAnodeAlignTableAxisX.monitoring.posRelative := FALSE;
   cmAnodeAlignTableAxisX.monitoring.posAbsolute := FALSE;
   cmAnodeAlignTableAxisX.monitoring.posSuperimposed := FALSE;
   cmAnodeAlignTableAxisX.monitoring.haltSuperimposed := FALSE;
   cmAnodeAlignTableAxisX.monitoring.brakeOpened := FALSE;
   cmAnodeAlignTableAxisX.monitoring.axisEnabled := TRUE;
   cmAnodeAlignTableAxisX.monitoring.resetActive := FALSE;
   cmAnodeAlignTableAxisX.monitoring.inVelocity := FALSE;
   cmAnodeAlignTableAxisX.monitoring.inLimitation := FALSE;
   cmAnodeAlignTableAxisX.monitoring.inClamping := FALSE;
   cmAnodeAlignTableAxisX.monitoring.startSync := FALSE;
   cmAnodeAlignTableAxisX.monitoring.inSync := FALSE;
   cmAnodeAlignTableAxisX.monitoring.inSimulation := FALSE;
   cmAnodeAlignTableAxisX.monitoring.jogSelected := FALSE;
   cmAnodeAlignTableAxisX.monitoring.moveVelocitySelected := FALSE;
   cmAnodeAlignTableAxisX.monitoring.stopSelected := FALSE;
   cmAnodeAlignTableAxisX.monitoring.fastStopSelected := FALSE;
   cmAnodeAlignTableAxisX.monitoring.torqueLimitingSelected := FALSE;
   cmAnodeAlignTableAxisX.monitoring.homingSelected := FALSE;
   cmAnodeAlignTableAxisX.monitoring.posRelativeSelected := FALSE;
   cmAnodeAlignTableAxisX.monitoring.posAbsoluteSelected := FALSE;
   cmAnodeAlignTableAxisX.monitoring.posSuperimposedSelected := FALSE;
   cmAnodeAlignTableAxisX.monitoring.haltSuperimposedSelected := FALSE;
   cmAnodeAlignTableAxisX.monitoring.commandBusy := FALSE;
   cmAnodeAlignTableAxisX.monitoring.commandDone := FALSE;
   cmAnodeAlignTableAxisX.monitoring.commandAborted := FALSE;
   cmAnodeAlignTableAxisX.monitoring.homingCommandBusy := FALSE;
   cmAnodeAlignTableAxisX.monitoring.homingCommandDone := FALSE;
   cmAnodeAlignTableAxisX.monitoring.homingCommandAborted := FALSE;
   cmAnodeAlignTableAxisX.monitoring.superimposedBusy := FALSE;
   cmAnodeAlignTableAxisX.monitoring.superimposedDone := FALSE;
   cmAnodeAlignTableAxisX.monitoring.superimposedAborted := FALSE;
   cmAnodeAlignTableAxisX.monitoring.selectSetPosition := -1;
   cmAnodeAlignTableAxisX.monitoring.selectionController := FALSE;
   cmAnodeAlignTableAxisX.monitoring.interlockGeneral := TRUE;
   cmAnodeAlignTableAxisX.monitoring.interlockJogForward := TRUE;
   cmAnodeAlignTableAxisX.monitoring.interlockJogBackward := TRUE;
   cmAnodeAlignTableAxisX.monitoring.interlockWarningGeneral := FALSE;
   cmAnodeAlignTableAxisX.monitoring.interlockWarningJogForward := FALSE;
   cmAnodeAlignTableAxisX.monitoring.interlockWarningJogBackward := FALSE;
   cmAnodeAlignTableAxisX.monitoring.valid := TRUE;
   cmAnodeAlignTableAxisX.monitoring.busy := TRUE;
   cmAnodeAlignTableAxisX.monitoring.error := FALSE;
   cmAnodeAlignTableAxisX.monitoring.status := 16#7002;
   cmAnodeAlignTableAxisX.monitoring.subfunctionStatus := 16#0000;
   cmAnodeAlignTableAxisX.monitoring.actualPosition := 0.0;
   cmAnodeAlignTableAxisX.monitoring.actualSpeed := 0.0;
   cmAnodeAlignTableAxisX.monitoring.speedUnit := 1062;
   cmAnodeAlignTableAxisX.monitoring.positionUnit := 1013;
   cmAnodeAlignTableAxisX.monitoring.axisStatus1 := 16#0200_10E1;
   cmAnodeAlignTableAxisX.monitoring.axisStatus2 := 16#0000_0000;
   cmAnodeAlignTableAxisX.monitoring.axisType := 1;
   cmAnodeAlignTableAxisX.monitoring.maxVelocity := 2500.0;
   cmAnodeAlignTableAxisX.monitoring.actualCurrent := 0.0;
   cmAnodeAlignTableAxisX.monitoring.actualTorque := 0.0;
   cmAnodeAlignTableAxisX.monitoring.velocityOverrideEnabled := FALSE;
   cmAnodeAlignTableAxisX.monitoring.sinaParaError := FALSE;
   cmAnodeAlignTableAxisX.monitoring.sinaParaStatus := 16#0000_0000;
   cmAnodeAlignTableAxisX.configuration.referenceDesignator := WSTRING#'AnodeAlignTableAxisX';
   cmAnodeAlignTableAxisX.configuration.disableAlarms := FALSE;
   cmAnodeAlignTableAxisX.configuration.masterControlPopUp := TRUE;
   cmAnodeAlignTableAxisX.configuration.setPositions[0].position := 0.0;
   cmAnodeAlignTableAxisX.configuration.setPositions[1].position := 1.0;
   cmAnodeAlignTableAxisX.configuration.setPositions[2..3].position := -4.08;
   cmAnodeAlignTableAxisX.configuration.setPositions[4].position := -2.08;
   cmAnodeAlignTableAxisX.configuration.setPositions[5..7].position := -0.08;
   cmAnodeAlignTableAxisX.configuration.setPositions[8].position := -2.08;
   cmAnodeAlignTableAxisX.configuration.setPositions[9].position := -4.08;
   cmAnodeAlignTableAxisX.configuration.setPositions[10].position := 8.5;
   cmAnodeAlignTableAxisX.configuration.setPositions[11..15].position := 0.0;
   cmAnodeAlignTableAxisX.configuration.setPositions[0..1].velocity := 50.0;
   cmAnodeAlignTableAxisX.configuration.setPositions[2..9].velocity := 30.0;
   cmAnodeAlignTableAxisX.configuration.setPositions[10..15].velocity := -1.0;
   cmAnodeAlignTableAxisX.configuration.setPositions[0..1].acceleration := 500.0;
   cmAnodeAlignTableAxisX.configuration.setPositions[2..9].acceleration := 30.0;
   cmAnodeAlignTableAxisX.configuration.setPositions[10..15].acceleration := -1.0;
   cmAnodeAlignTableAxisX.configuration.setPositions[0..1].deceleration := 500.0;
   cmAnodeAlignTableAxisX.configuration.setPositions[2..9].deceleration := 30.0;
   cmAnodeAlignTableAxisX.configuration.setPositions[10..15].deceleration := -1.0;
   cmAnodeAlignTableAxisX.configuration.setPositions[0..15]."name" := '';
   cmAnodeAlignTableAxisY1.commandConfiguration.generalSettings.stopOnError := TRUE;
   cmAnodeAlignTableAxisY1.commandConfiguration.generalSettings.resetWithRestart := FALSE;
   cmAnodeAlignTableAxisY1.commandConfiguration.generalSettings.abortWaitingSyncCmd := TRUE;
   cmAnodeAlignTableAxisY1.commandConfiguration.power.startMode := 1;
   cmAnodeAlignTableAxisY1.commandConfiguration.power.stopMode := 0;
   cmAnodeAlignTableAxisY1.commandConfiguration.power.syncMotionSimulation := FALSE;
   cmAnodeAlignTableAxisY1.commandConfiguration.power.syncMotionSimulationExtendedMode := -1;
   cmAnodeAlignTableAxisY1.commandConfiguration.jog.velocity := 10.0;
   cmAnodeAlignTableAxisY1.commandConfiguration.jog.acceleration := 100.0;
   cmAnodeAlignTableAxisY1.commandConfiguration.jog.deceleration := 100.0;
   cmAnodeAlignTableAxisY1.commandConfiguration.jog.jerk := -1.0;
   cmAnodeAlignTableAxisY1.commandConfiguration.jog.positionControlled := TRUE;
   cmAnodeAlignTableAxisY1.commandConfiguration.jog.increment := 0.0;
   cmAnodeAlignTableAxisY1.commandConfiguration.jog.mode := 0;
   cmAnodeAlignTableAxisY1.commandConfiguration.moveVelocity.velocity := 10.0;
   cmAnodeAlignTableAxisY1.commandConfiguration.moveVelocity.acceleration := 100.0;
   cmAnodeAlignTableAxisY1.commandConfiguration.moveVelocity.deceleration := 100.0;
   cmAnodeAlignTableAxisY1.commandConfiguration.moveVelocity.jerk := -1.0;
   cmAnodeAlignTableAxisY1.commandConfiguration.moveVelocity.direction := 0;
   cmAnodeAlignTableAxisY1.commandConfiguration.moveVelocity.positionControlled := TRUE;
   cmAnodeAlignTableAxisY1.commandConfiguration.moveVelocity.velocityChangeOnTheFly := FALSE;
   cmAnodeAlignTableAxisY1.commandConfiguration.stop.deceleration := -1.0;
   cmAnodeAlignTableAxisY1.commandConfiguration.stop.jerk := -1.0;
   cmAnodeAlignTableAxisY1.commandConfiguration.stop.abortAcceleration := FALSE;
   cmAnodeAlignTableAxisY1.commandConfiguration.fastStop.deceleration := -1.0;
   cmAnodeAlignTableAxisY1.commandConfiguration.fastStop.jerk := -1.0;
   cmAnodeAlignTableAxisY1.commandConfiguration.fastStop.abortAcceleration := FALSE;
   cmAnodeAlignTableAxisY1.commandConfiguration.fastStop.replaceStopPossible := FALSE;
   cmAnodeAlignTableAxisY1.commandConfiguration.torqueLimiting.limit := -1.0;
   cmAnodeAlignTableAxisY1.commandConfiguration.torqueLimiting.mode := 0;
   cmAnodeAlignTableAxisY1.commandConfiguration.homing.position := 0.0;
   cmAnodeAlignTableAxisY1.commandConfiguration.homing.mode := 0;
   cmAnodeAlignTableAxisY1.commandConfiguration.homing.sensor := 0;
   cmAnodeAlignTableAxisY1.commandConfiguration.homing.extendedMode := -1;
   cmAnodeAlignTableAxisY1.commandConfiguration.homing.extendedModeTorqueLimit := 0.0;
   cmAnodeAlignTableAxisY1.commandConfiguration.homing.extendedModeTargetPosition := 0.0;
   cmAnodeAlignTableAxisY1.commandConfiguration.posRelative.distance := 0.0;
   cmAnodeAlignTableAxisY1.commandConfiguration.posRelative.velocity := 10.0;
   cmAnodeAlignTableAxisY1.commandConfiguration.posRelative.acceleration := 100.0;
   cmAnodeAlignTableAxisY1.commandConfiguration.posRelative.deceleration := 100.0;
   cmAnodeAlignTableAxisY1.commandConfiguration.posRelative.jerk := -1.0;
   cmAnodeAlignTableAxisY1.commandConfiguration.posRelative.direction := 0;
   cmAnodeAlignTableAxisY1.commandConfiguration.posAbsolute.position := 0.0;
   cmAnodeAlignTableAxisY1.commandConfiguration.posAbsolute.velocity := -1.0;
   cmAnodeAlignTableAxisY1.commandConfiguration.posAbsolute.acceleration := -1.0;
   cmAnodeAlignTableAxisY1.commandConfiguration.posAbsolute.deceleration := -1.0;
   cmAnodeAlignTableAxisY1.commandConfiguration.posAbsolute.jerk := -1.0;
   cmAnodeAlignTableAxisY1.commandConfiguration.posAbsolute.direction := 1;
   cmAnodeAlignTableAxisY1.commandConfiguration.posAbsolute.positionChangeOnTheFly := FALSE;
   cmAnodeAlignTableAxisY1.commandConfiguration.posAbsolute.velocityChangeOnTheFly := FALSE;
   cmAnodeAlignTableAxisY1.commandConfiguration.posSuperimposed.distance := 0.0;
   cmAnodeAlignTableAxisY1.commandConfiguration.posSuperimposed.velocityDiff := -1.0;
   cmAnodeAlignTableAxisY1.commandConfiguration.posSuperimposed.acceleration := -1.0;
   cmAnodeAlignTableAxisY1.commandConfiguration.posSuperimposed.deceleration := -1.0;
   cmAnodeAlignTableAxisY1.commandConfiguration.posSuperimposed.jerk := -1.0;
   cmAnodeAlignTableAxisY1.commandConfiguration.posSuperimposed.direction := 0;
   cmAnodeAlignTableAxisY1.commandConfiguration.haltSuperimposed.deceleration := -1.0;
   cmAnodeAlignTableAxisY1.commandConfiguration.haltSuperimposed.jerk := -1.0;
   cmAnodeAlignTableAxisY1.commandConfiguration.haltSuperimposed.abortAcceleration := FALSE;
   cmAnodeAlignTableAxisY1.commandConfiguration.gearInRelative.ratioNumerator := 1;
   cmAnodeAlignTableAxisY1.commandConfiguration.gearInRelative.ratioDenominator := 1;
   cmAnodeAlignTableAxisY1.commandConfiguration.gearInRelative.acceleration := -1.0;
   cmAnodeAlignTableAxisY1.commandConfiguration.gearInRelative.deceleration := -1.0;
   cmAnodeAlignTableAxisY1.commandConfiguration.gearInRelative.jerk := -1.0;
   cmAnodeAlignTableAxisY1.commandConfiguration.gearInRelative.ratioChangeOnTheFly := FALSE;
   cmAnodeAlignTableAxisY1.commandConfiguration.gearInAbsolute.ratioNumerator := 1;
   cmAnodeAlignTableAxisY1.commandConfiguration.gearInAbsolute.ratioDenominator := 1;
   cmAnodeAlignTableAxisY1.commandConfiguration.gearInAbsolute.masterSyncPosition := 0.0;
   cmAnodeAlignTableAxisY1.commandConfiguration.gearInAbsolute.slaveSyncPosition := 0.0;
   cmAnodeAlignTableAxisY1.commandConfiguration.gearInAbsolute.syncProfileReference := 1;
   cmAnodeAlignTableAxisY1.commandConfiguration.gearInAbsolute.masterStartDistance := 0.0;
   cmAnodeAlignTableAxisY1.commandConfiguration.gearInAbsolute.velocity := -1.0;
   cmAnodeAlignTableAxisY1.commandConfiguration.gearInAbsolute.acceleration := -1.0;
   cmAnodeAlignTableAxisY1.commandConfiguration.gearInAbsolute.deceleration := -1.0;
   cmAnodeAlignTableAxisY1.commandConfiguration.gearInAbsolute.jerk := -1.0;
   cmAnodeAlignTableAxisY1.commandConfiguration.gearInAbsolute.syncDirection := 1;
   cmAnodeAlignTableAxisY1.commandConfiguration.gearInAbsolute.ratioChangeOnTheFly := FALSE;
   cmAnodeAlignTableAxisY1.commandConfiguration.gearInVelocity.continuousUpdate := FALSE;
   cmAnodeAlignTableAxisY1.commandConfiguration.gearInVelocity.ratioNumerator := 1;
   cmAnodeAlignTableAxisY1.commandConfiguration.gearInVelocity.ratioDenominator := 1;
   cmAnodeAlignTableAxisY1.commandConfiguration.gearInVelocity.acceleration := -1.0;
   cmAnodeAlignTableAxisY1.commandConfiguration.gearInVelocity.deceleration := -1.0;
   cmAnodeAlignTableAxisY1.commandConfiguration.gearInVelocity.jerk := -1.0;
   cmAnodeAlignTableAxisY1.commandConfiguration.gearInVelocity.positionControlled := FALSE;
   cmAnodeAlignTableAxisY1.commandConfiguration.camIn.masterOffset := 0.0;
   cmAnodeAlignTableAxisY1.commandConfiguration.camIn.slaveOffset := 0.0;
   cmAnodeAlignTableAxisY1.commandConfiguration.camIn.masterScaling := 1.0;
   cmAnodeAlignTableAxisY1.commandConfiguration.camIn.slaveScaling := 1.0;
   cmAnodeAlignTableAxisY1.commandConfiguration.camIn.masterSyncPosition := 0.0;
   cmAnodeAlignTableAxisY1.commandConfiguration.camIn.syncProfileReference := 1;
   cmAnodeAlignTableAxisY1.commandConfiguration.camIn.masterStartDistance := 0.0;
   cmAnodeAlignTableAxisY1.commandConfiguration.camIn.velocity := -1.0;
   cmAnodeAlignTableAxisY1.commandConfiguration.camIn.acceleration := -1.0;
   cmAnodeAlignTableAxisY1.commandConfiguration.camIn.deceleration := -1.0;
   cmAnodeAlignTableAxisY1.commandConfiguration.camIn.jerk := -1.0;
   cmAnodeAlignTableAxisY1.commandConfiguration.camIn.applicationMode := 0;
   cmAnodeAlignTableAxisY1.commandConfiguration.camIn.syncDirection := 1;
   cmAnodeAlignTableAxisY1.commandConfiguration.gearOutCamOut.slavePosition := 0.0;
   cmAnodeAlignTableAxisY1.commandConfiguration.gearOutCamOut.syncProfileReference := 1;
   cmAnodeAlignTableAxisY1.commandConfiguration.gearOutCamOut.masterStopDistance := 0.0;
   cmAnodeAlignTableAxisY1.commandConfiguration.gearOutCamOut.deceleration := -1.0;
   cmAnodeAlignTableAxisY1.commandConfiguration.gearOutCamOut.jerk := -1.0;
   cmAnodeAlignTableAxisY1.commandConfiguration.gearOutCamOut.syncOutDirection := 3;
   cmAnodeAlignTableAxisY1.commandConfiguration.gearOutCamOut.gearOutCamOutMode := -1;
   cmAnodeAlignTableAxisY1.commandConfiguration.phasing.phaseShift := 0.0;
   cmAnodeAlignTableAxisY1.commandConfiguration.phasing.velocity := -1.0;
   cmAnodeAlignTableAxisY1.commandConfiguration.phasing.acceleration := -1.0;
   cmAnodeAlignTableAxisY1.commandConfiguration.phasing.deceleration := -1.0;
   cmAnodeAlignTableAxisY1.commandConfiguration.phasing.jerk := -1.0;
   cmAnodeAlignTableAxisY1.commandConfiguration.phasing.profileReference := 0;
   cmAnodeAlignTableAxisY1.commandConfiguration.phasing.phasingDistance := 0.0;
   cmAnodeAlignTableAxisY1.commandConfiguration.phasing.startPosition := 0.0;
   cmAnodeAlignTableAxisY1.commandConfiguration.phasing.direction := 3;
   cmAnodeAlignTableAxisY1.commandConfiguration.phasing.phaseAbsolute := TRUE;
   cmAnodeAlignTableAxisY1.commandConfiguration.phasing.phaseShiftChangeOnTheFly := FALSE;
   cmAnodeAlignTableAxisY1.commandConfiguration.offset.offset := 0.0;
   cmAnodeAlignTableAxisY1.commandConfiguration.offset.profileReference := 1;
   cmAnodeAlignTableAxisY1.commandConfiguration.offset.offsetDistance := 0.0;
   cmAnodeAlignTableAxisY1.commandConfiguration.offset.startPosition := 0.0;
   cmAnodeAlignTableAxisY1.commandConfiguration.offset.direction := 3;
   cmAnodeAlignTableAxisY1.commandConfiguration.offset.offsetAbsolute := TRUE;
   cmAnodeAlignTableAxisY1.commandConfiguration.offset.offsetChangeOnTheFly := FALSE;
   cmAnodeAlignTableAxisY1.commands.enableMasterControl := TRUE;
   cmAnodeAlignTableAxisY1.commands.enableAxis := FALSE;
   cmAnodeAlignTableAxisY1.commands.resetAxis := FALSE;
   cmAnodeAlignTableAxisY1.commands.openBrake := FALSE;
   cmAnodeAlignTableAxisY1.commands.jogForward := FALSE;
   cmAnodeAlignTableAxisY1.commands.jogBackward := FALSE;
   cmAnodeAlignTableAxisY1.commands.moveVelocity := FALSE;
   cmAnodeAlignTableAxisY1.commands.stop := FALSE;
   cmAnodeAlignTableAxisY1.commands.fastStop := FALSE;
   cmAnodeAlignTableAxisY1.commands.torqueLimiting := FALSE;
   cmAnodeAlignTableAxisY1.commands.homing := FALSE;
   cmAnodeAlignTableAxisY1.commands.posRelative := FALSE;
   cmAnodeAlignTableAxisY1.commands.posAbsolute := FALSE;
   cmAnodeAlignTableAxisY1.commands.posSuperimposed := FALSE;
   cmAnodeAlignTableAxisY1.commands.haltSuperimposed := FALSE;
   cmAnodeAlignTableAxisY1.commands.selectSetPosition := -1;
   cmAnodeAlignTableAxisY1.commands.uploadParameters := FALSE;
   cmAnodeAlignTableAxisY1.commands.refreshConfiguration := FALSE;
   cmAnodeAlignTableAxisY1.commands.editConfiguration := FALSE;
   cmAnodeAlignTableAxisY1.commands.saveConfiguration := FALSE;
   cmAnodeAlignTableAxisY1.commands.uploadCurrentTorque := FALSE;
   cmAnodeAlignTableAxisY1.commands.reset := FALSE;
   cmAnodeAlignTableAxisY1.monitoring.enable := TRUE;
   cmAnodeAlignTableAxisY1.monitoring.referenceDesignator := WSTRING#'AnodeAlignTableAxisY1';
   cmAnodeAlignTableAxisY1.monitoring.enabled := TRUE;
   cmAnodeAlignTableAxisY1.monitoring.enableManualCmds := FALSE;
   cmAnodeAlignTableAxisY1.monitoring.reset := FALSE;
   cmAnodeAlignTableAxisY1.monitoring.resetAxis := FALSE;
   cmAnodeAlignTableAxisY1.monitoring.enableAxis := TRUE;
   cmAnodeAlignTableAxisY1.monitoring.openBrake := FALSE;
   cmAnodeAlignTableAxisY1.monitoring.jogBackward := FALSE;
   cmAnodeAlignTableAxisY1.monitoring.jogForward := FALSE;
   cmAnodeAlignTableAxisY1.monitoring.moveVelocity := FALSE;
   cmAnodeAlignTableAxisY1.monitoring.stop := FALSE;
   cmAnodeAlignTableAxisY1.monitoring.fastStop := FALSE;
   cmAnodeAlignTableAxisY1.monitoring.torqueLimiting := FALSE;
   cmAnodeAlignTableAxisY1.monitoring.homing := FALSE;
   cmAnodeAlignTableAxisY1.monitoring.posRelative := FALSE;
   cmAnodeAlignTableAxisY1.monitoring.posAbsolute := FALSE;
   cmAnodeAlignTableAxisY1.monitoring.posSuperimposed := FALSE;
   cmAnodeAlignTableAxisY1.monitoring.haltSuperimposed := FALSE;
   cmAnodeAlignTableAxisY1.monitoring.brakeOpened := FALSE;
   cmAnodeAlignTableAxisY1.monitoring.axisEnabled := TRUE;
   cmAnodeAlignTableAxisY1.monitoring.resetActive := FALSE;
   cmAnodeAlignTableAxisY1.monitoring.inVelocity := FALSE;
   cmAnodeAlignTableAxisY1.monitoring.inLimitation := FALSE;
   cmAnodeAlignTableAxisY1.monitoring.inClamping := FALSE;
   cmAnodeAlignTableAxisY1.monitoring.startSync := FALSE;
   cmAnodeAlignTableAxisY1.monitoring.inSync := FALSE;
   cmAnodeAlignTableAxisY1.monitoring.inSimulation := FALSE;
   cmAnodeAlignTableAxisY1.monitoring.jogSelected := FALSE;
   cmAnodeAlignTableAxisY1.monitoring.moveVelocitySelected := FALSE;
   cmAnodeAlignTableAxisY1.monitoring.stopSelected := FALSE;
   cmAnodeAlignTableAxisY1.monitoring.fastStopSelected := FALSE;
   cmAnodeAlignTableAxisY1.monitoring.torqueLimitingSelected := FALSE;
   cmAnodeAlignTableAxisY1.monitoring.homingSelected := FALSE;
   cmAnodeAlignTableAxisY1.monitoring.posRelativeSelected := FALSE;
   cmAnodeAlignTableAxisY1.monitoring.posAbsoluteSelected := FALSE;
   cmAnodeAlignTableAxisY1.monitoring.posSuperimposedSelected := FALSE;
   cmAnodeAlignTableAxisY1.monitoring.haltSuperimposedSelected := FALSE;
   cmAnodeAlignTableAxisY1.monitoring.commandBusy := FALSE;
   cmAnodeAlignTableAxisY1.monitoring.commandDone := FALSE;
   cmAnodeAlignTableAxisY1.monitoring.commandAborted := FALSE;
   cmAnodeAlignTableAxisY1.monitoring.homingCommandBusy := FALSE;
   cmAnodeAlignTableAxisY1.monitoring.homingCommandDone := FALSE;
   cmAnodeAlignTableAxisY1.monitoring.homingCommandAborted := FALSE;
   cmAnodeAlignTableAxisY1.monitoring.superimposedBusy := FALSE;
   cmAnodeAlignTableAxisY1.monitoring.superimposedDone := FALSE;
   cmAnodeAlignTableAxisY1.monitoring.superimposedAborted := FALSE;
   cmAnodeAlignTableAxisY1.monitoring.selectSetPosition := -1;
   cmAnodeAlignTableAxisY1.monitoring.selectionController := FALSE;
   cmAnodeAlignTableAxisY1.monitoring.interlockGeneral := TRUE;
   cmAnodeAlignTableAxisY1.monitoring.interlockJogForward := TRUE;
   cmAnodeAlignTableAxisY1.monitoring.interlockJogBackward := TRUE;
   cmAnodeAlignTableAxisY1.monitoring.interlockWarningGeneral := FALSE;
   cmAnodeAlignTableAxisY1.monitoring.interlockWarningJogForward := FALSE;
   cmAnodeAlignTableAxisY1.monitoring.interlockWarningJogBackward := FALSE;
   cmAnodeAlignTableAxisY1.monitoring.valid := TRUE;
   cmAnodeAlignTableAxisY1.monitoring.busy := TRUE;
   cmAnodeAlignTableAxisY1.monitoring.error := FALSE;
   cmAnodeAlignTableAxisY1.monitoring.status := 16#7002;
   cmAnodeAlignTableAxisY1.monitoring.subfunctionStatus := 16#0000;
   cmAnodeAlignTableAxisY1.monitoring.actualPosition := 0.0;
   cmAnodeAlignTableAxisY1.monitoring.actualSpeed := 0.0;
   cmAnodeAlignTableAxisY1.monitoring.speedUnit := 1062;
   cmAnodeAlignTableAxisY1.monitoring.positionUnit := 1013;
   cmAnodeAlignTableAxisY1.monitoring.axisStatus1 := 16#0200_10E1;
   cmAnodeAlignTableAxisY1.monitoring.axisStatus2 := 16#0000_0000;
   cmAnodeAlignTableAxisY1.monitoring.axisType := 1;
   cmAnodeAlignTableAxisY1.monitoring.maxVelocity := 2500.0;
   cmAnodeAlignTableAxisY1.monitoring.actualCurrent := 0.0;
   cmAnodeAlignTableAxisY1.monitoring.actualTorque := 0.0;
   cmAnodeAlignTableAxisY1.monitoring.velocityOverrideEnabled := FALSE;
   cmAnodeAlignTableAxisY1.monitoring.sinaParaError := FALSE;
   cmAnodeAlignTableAxisY1.monitoring.sinaParaStatus := 16#0000_0000;
   cmAnodeAlignTableAxisY1.configuration.referenceDesignator := WSTRING#'AnodeAlignTableAxisY1';
   cmAnodeAlignTableAxisY1.configuration.disableAlarms := FALSE;
   cmAnodeAlignTableAxisY1.configuration.masterControlPopUp := TRUE;
   cmAnodeAlignTableAxisY1.configuration.setPositions[0].position := 0.0;
   cmAnodeAlignTableAxisY1.configuration.setPositions[1].position := 2.0;
   cmAnodeAlignTableAxisY1.configuration.setPositions[2].position := 0.6;
   cmAnodeAlignTableAxisY1.configuration.setPositions[3..5].position := 2.6;
   cmAnodeAlignTableAxisY1.configuration.setPositions[6].position := 0.6;
   cmAnodeAlignTableAxisY1.configuration.setPositions[7].position := -1.4;
   cmAnodeAlignTableAxisY1.configuration.setPositions[8].position := 0.6;
   cmAnodeAlignTableAxisY1.configuration.setPositions[9].position := -1.4;
   cmAnodeAlignTableAxisY1.configuration.setPositions[10].position := 8.5;
   cmAnodeAlignTableAxisY1.configuration.setPositions[11..15].position := 0.0;
   cmAnodeAlignTableAxisY1.configuration.setPositions[0..1].velocity := 50.0;
   cmAnodeAlignTableAxisY1.configuration.setPositions[2..9].velocity := 30.0;
   cmAnodeAlignTableAxisY1.configuration.setPositions[10..15].velocity := -1.0;
   cmAnodeAlignTableAxisY1.configuration.setPositions[0..1].acceleration := 500.0;
   cmAnodeAlignTableAxisY1.configuration.setPositions[2..9].acceleration := 30.0;
   cmAnodeAlignTableAxisY1.configuration.setPositions[10..15].acceleration := -1.0;
   cmAnodeAlignTableAxisY1.configuration.setPositions[0..1].deceleration := 500.0;
   cmAnodeAlignTableAxisY1.configuration.setPositions[2..9].deceleration := 30.0;
   cmAnodeAlignTableAxisY1.configuration.setPositions[10..15].deceleration := -1.0;
   cmAnodeAlignTableAxisY1.configuration.setPositions[0..15]."name" := '';
   cmAnodeAlignTableAxisY2.commandConfiguration.generalSettings.stopOnError := TRUE;
   cmAnodeAlignTableAxisY2.commandConfiguration.generalSettings.resetWithRestart := FALSE;
   cmAnodeAlignTableAxisY2.commandConfiguration.generalSettings.abortWaitingSyncCmd := TRUE;
   cmAnodeAlignTableAxisY2.commandConfiguration.power.startMode := 1;
   cmAnodeAlignTableAxisY2.commandConfiguration.power.stopMode := 0;
   cmAnodeAlignTableAxisY2.commandConfiguration.power.syncMotionSimulation := FALSE;
   cmAnodeAlignTableAxisY2.commandConfiguration.power.syncMotionSimulationExtendedMode := -1;
   cmAnodeAlignTableAxisY2.commandConfiguration.jog.velocity := 10.0;
   cmAnodeAlignTableAxisY2.commandConfiguration.jog.acceleration := 100.0;
   cmAnodeAlignTableAxisY2.commandConfiguration.jog.deceleration := 100.0;
   cmAnodeAlignTableAxisY2.commandConfiguration.jog.jerk := -1.0;
   cmAnodeAlignTableAxisY2.commandConfiguration.jog.positionControlled := TRUE;
   cmAnodeAlignTableAxisY2.commandConfiguration.jog.increment := 0.0;
   cmAnodeAlignTableAxisY2.commandConfiguration.jog.mode := 0;
   cmAnodeAlignTableAxisY2.commandConfiguration.moveVelocity.velocity := 10.0;
   cmAnodeAlignTableAxisY2.commandConfiguration.moveVelocity.acceleration := 100.0;
   cmAnodeAlignTableAxisY2.commandConfiguration.moveVelocity.deceleration := 100.0;
   cmAnodeAlignTableAxisY2.commandConfiguration.moveVelocity.jerk := -1.0;
   cmAnodeAlignTableAxisY2.commandConfiguration.moveVelocity.direction := 0;
   cmAnodeAlignTableAxisY2.commandConfiguration.moveVelocity.positionControlled := TRUE;
   cmAnodeAlignTableAxisY2.commandConfiguration.moveVelocity.velocityChangeOnTheFly := FALSE;
   cmAnodeAlignTableAxisY2.commandConfiguration.stop.deceleration := -1.0;
   cmAnodeAlignTableAxisY2.commandConfiguration.stop.jerk := -1.0;
   cmAnodeAlignTableAxisY2.commandConfiguration.stop.abortAcceleration := FALSE;
   cmAnodeAlignTableAxisY2.commandConfiguration.fastStop.deceleration := -1.0;
   cmAnodeAlignTableAxisY2.commandConfiguration.fastStop.jerk := -1.0;
   cmAnodeAlignTableAxisY2.commandConfiguration.fastStop.abortAcceleration := FALSE;
   cmAnodeAlignTableAxisY2.commandConfiguration.fastStop.replaceStopPossible := FALSE;
   cmAnodeAlignTableAxisY2.commandConfiguration.torqueLimiting.limit := -1.0;
   cmAnodeAlignTableAxisY2.commandConfiguration.torqueLimiting.mode := 0;
   cmAnodeAlignTableAxisY2.commandConfiguration.homing.position := 0.0;
   cmAnodeAlignTableAxisY2.commandConfiguration.homing.mode := 0;
   cmAnodeAlignTableAxisY2.commandConfiguration.homing.sensor := 0;
   cmAnodeAlignTableAxisY2.commandConfiguration.homing.extendedMode := -1;
   cmAnodeAlignTableAxisY2.commandConfiguration.homing.extendedModeTorqueLimit := 0.0;
   cmAnodeAlignTableAxisY2.commandConfiguration.homing.extendedModeTargetPosition := 0.0;
   cmAnodeAlignTableAxisY2.commandConfiguration.posRelative.distance := 0.0;
   cmAnodeAlignTableAxisY2.commandConfiguration.posRelative.velocity := 10.0;
   cmAnodeAlignTableAxisY2.commandConfiguration.posRelative.acceleration := 100.0;
   cmAnodeAlignTableAxisY2.commandConfiguration.posRelative.deceleration := 100.0;
   cmAnodeAlignTableAxisY2.commandConfiguration.posRelative.jerk := -1.0;
   cmAnodeAlignTableAxisY2.commandConfiguration.posRelative.direction := 0;
   cmAnodeAlignTableAxisY2.commandConfiguration.posAbsolute.position := 0.0;
   cmAnodeAlignTableAxisY2.commandConfiguration.posAbsolute.velocity := -1.0;
   cmAnodeAlignTableAxisY2.commandConfiguration.posAbsolute.acceleration := -1.0;
   cmAnodeAlignTableAxisY2.commandConfiguration.posAbsolute.deceleration := -1.0;
   cmAnodeAlignTableAxisY2.commandConfiguration.posAbsolute.jerk := -1.0;
   cmAnodeAlignTableAxisY2.commandConfiguration.posAbsolute.direction := 1;
   cmAnodeAlignTableAxisY2.commandConfiguration.posAbsolute.positionChangeOnTheFly := FALSE;
   cmAnodeAlignTableAxisY2.commandConfiguration.posAbsolute.velocityChangeOnTheFly := FALSE;
   cmAnodeAlignTableAxisY2.commandConfiguration.posSuperimposed.distance := 0.0;
   cmAnodeAlignTableAxisY2.commandConfiguration.posSuperimposed.velocityDiff := -1.0;
   cmAnodeAlignTableAxisY2.commandConfiguration.posSuperimposed.acceleration := -1.0;
   cmAnodeAlignTableAxisY2.commandConfiguration.posSuperimposed.deceleration := -1.0;
   cmAnodeAlignTableAxisY2.commandConfiguration.posSuperimposed.jerk := -1.0;
   cmAnodeAlignTableAxisY2.commandConfiguration.posSuperimposed.direction := 0;
   cmAnodeAlignTableAxisY2.commandConfiguration.haltSuperimposed.deceleration := -1.0;
   cmAnodeAlignTableAxisY2.commandConfiguration.haltSuperimposed.jerk := -1.0;
   cmAnodeAlignTableAxisY2.commandConfiguration.haltSuperimposed.abortAcceleration := FALSE;
   cmAnodeAlignTableAxisY2.commandConfiguration.gearInRelative.ratioNumerator := 1;
   cmAnodeAlignTableAxisY2.commandConfiguration.gearInRelative.ratioDenominator := 1;
   cmAnodeAlignTableAxisY2.commandConfiguration.gearInRelative.acceleration := -1.0;
   cmAnodeAlignTableAxisY2.commandConfiguration.gearInRelative.deceleration := -1.0;
   cmAnodeAlignTableAxisY2.commandConfiguration.gearInRelative.jerk := -1.0;
   cmAnodeAlignTableAxisY2.commandConfiguration.gearInRelative.ratioChangeOnTheFly := FALSE;
   cmAnodeAlignTableAxisY2.commandConfiguration.gearInAbsolute.ratioNumerator := 1;
   cmAnodeAlignTableAxisY2.commandConfiguration.gearInAbsolute.ratioDenominator := 1;
   cmAnodeAlignTableAxisY2.commandConfiguration.gearInAbsolute.masterSyncPosition := 0.0;
   cmAnodeAlignTableAxisY2.commandConfiguration.gearInAbsolute.slaveSyncPosition := 0.0;
   cmAnodeAlignTableAxisY2.commandConfiguration.gearInAbsolute.syncProfileReference := 1;
   cmAnodeAlignTableAxisY2.commandConfiguration.gearInAbsolute.masterStartDistance := 0.0;
   cmAnodeAlignTableAxisY2.commandConfiguration.gearInAbsolute.velocity := -1.0;
   cmAnodeAlignTableAxisY2.commandConfiguration.gearInAbsolute.acceleration := -1.0;
   cmAnodeAlignTableAxisY2.commandConfiguration.gearInAbsolute.deceleration := -1.0;
   cmAnodeAlignTableAxisY2.commandConfiguration.gearInAbsolute.jerk := -1.0;
   cmAnodeAlignTableAxisY2.commandConfiguration.gearInAbsolute.syncDirection := 1;
   cmAnodeAlignTableAxisY2.commandConfiguration.gearInAbsolute.ratioChangeOnTheFly := FALSE;
   cmAnodeAlignTableAxisY2.commandConfiguration.gearInVelocity.continuousUpdate := FALSE;
   cmAnodeAlignTableAxisY2.commandConfiguration.gearInVelocity.ratioNumerator := 1;
   cmAnodeAlignTableAxisY2.commandConfiguration.gearInVelocity.ratioDenominator := 1;
   cmAnodeAlignTableAxisY2.commandConfiguration.gearInVelocity.acceleration := -1.0;
   cmAnodeAlignTableAxisY2.commandConfiguration.gearInVelocity.deceleration := -1.0;
   cmAnodeAlignTableAxisY2.commandConfiguration.gearInVelocity.jerk := -1.0;
   cmAnodeAlignTableAxisY2.commandConfiguration.gearInVelocity.positionControlled := FALSE;
   cmAnodeAlignTableAxisY2.commandConfiguration.camIn.masterOffset := 0.0;
   cmAnodeAlignTableAxisY2.commandConfiguration.camIn.slaveOffset := 0.0;
   cmAnodeAlignTableAxisY2.commandConfiguration.camIn.masterScaling := 1.0;
   cmAnodeAlignTableAxisY2.commandConfiguration.camIn.slaveScaling := 1.0;
   cmAnodeAlignTableAxisY2.commandConfiguration.camIn.masterSyncPosition := 0.0;
   cmAnodeAlignTableAxisY2.commandConfiguration.camIn.syncProfileReference := 1;
   cmAnodeAlignTableAxisY2.commandConfiguration.camIn.masterStartDistance := 0.0;
   cmAnodeAlignTableAxisY2.commandConfiguration.camIn.velocity := -1.0;
   cmAnodeAlignTableAxisY2.commandConfiguration.camIn.acceleration := -1.0;
   cmAnodeAlignTableAxisY2.commandConfiguration.camIn.deceleration := -1.0;
   cmAnodeAlignTableAxisY2.commandConfiguration.camIn.jerk := -1.0;
   cmAnodeAlignTableAxisY2.commandConfiguration.camIn.applicationMode := 0;
   cmAnodeAlignTableAxisY2.commandConfiguration.camIn.syncDirection := 1;
   cmAnodeAlignTableAxisY2.commandConfiguration.gearOutCamOut.slavePosition := 0.0;
   cmAnodeAlignTableAxisY2.commandConfiguration.gearOutCamOut.syncProfileReference := 1;
   cmAnodeAlignTableAxisY2.commandConfiguration.gearOutCamOut.masterStopDistance := 0.0;
   cmAnodeAlignTableAxisY2.commandConfiguration.gearOutCamOut.deceleration := -1.0;
   cmAnodeAlignTableAxisY2.commandConfiguration.gearOutCamOut.jerk := -1.0;
   cmAnodeAlignTableAxisY2.commandConfiguration.gearOutCamOut.syncOutDirection := 3;
   cmAnodeAlignTableAxisY2.commandConfiguration.gearOutCamOut.gearOutCamOutMode := -1;
   cmAnodeAlignTableAxisY2.commandConfiguration.phasing.phaseShift := 0.0;
   cmAnodeAlignTableAxisY2.commandConfiguration.phasing.velocity := -1.0;
   cmAnodeAlignTableAxisY2.commandConfiguration.phasing.acceleration := -1.0;
   cmAnodeAlignTableAxisY2.commandConfiguration.phasing.deceleration := -1.0;
   cmAnodeAlignTableAxisY2.commandConfiguration.phasing.jerk := -1.0;
   cmAnodeAlignTableAxisY2.commandConfiguration.phasing.profileReference := 0;
   cmAnodeAlignTableAxisY2.commandConfiguration.phasing.phasingDistance := 0.0;
   cmAnodeAlignTableAxisY2.commandConfiguration.phasing.startPosition := 0.0;
   cmAnodeAlignTableAxisY2.commandConfiguration.phasing.direction := 3;
   cmAnodeAlignTableAxisY2.commandConfiguration.phasing.phaseAbsolute := TRUE;
   cmAnodeAlignTableAxisY2.commandConfiguration.phasing.phaseShiftChangeOnTheFly := FALSE;
   cmAnodeAlignTableAxisY2.commandConfiguration.offset.offset := 0.0;
   cmAnodeAlignTableAxisY2.commandConfiguration.offset.profileReference := 1;
   cmAnodeAlignTableAxisY2.commandConfiguration.offset.offsetDistance := 0.0;
   cmAnodeAlignTableAxisY2.commandConfiguration.offset.startPosition := 0.0;
   cmAnodeAlignTableAxisY2.commandConfiguration.offset.direction := 3;
   cmAnodeAlignTableAxisY2.commandConfiguration.offset.offsetAbsolute := TRUE;
   cmAnodeAlignTableAxisY2.commandConfiguration.offset.offsetChangeOnTheFly := FALSE;
   cmAnodeAlignTableAxisY2.commands.enableMasterControl := TRUE;
   cmAnodeAlignTableAxisY2.commands.enableAxis := FALSE;
   cmAnodeAlignTableAxisY2.commands.resetAxis := FALSE;
   cmAnodeAlignTableAxisY2.commands.openBrake := FALSE;
   cmAnodeAlignTableAxisY2.commands.jogForward := FALSE;
   cmAnodeAlignTableAxisY2.commands.jogBackward := FALSE;
   cmAnodeAlignTableAxisY2.commands.moveVelocity := FALSE;
   cmAnodeAlignTableAxisY2.commands.stop := FALSE;
   cmAnodeAlignTableAxisY2.commands.fastStop := FALSE;
   cmAnodeAlignTableAxisY2.commands.torqueLimiting := FALSE;
   cmAnodeAlignTableAxisY2.commands.homing := FALSE;
   cmAnodeAlignTableAxisY2.commands.posRelative := FALSE;
   cmAnodeAlignTableAxisY2.commands.posAbsolute := FALSE;
   cmAnodeAlignTableAxisY2.commands.posSuperimposed := FALSE;
   cmAnodeAlignTableAxisY2.commands.haltSuperimposed := FALSE;
   cmAnodeAlignTableAxisY2.commands.selectSetPosition := -1;
   cmAnodeAlignTableAxisY2.commands.uploadParameters := FALSE;
   cmAnodeAlignTableAxisY2.commands.refreshConfiguration := FALSE;
   cmAnodeAlignTableAxisY2.commands.editConfiguration := FALSE;
   cmAnodeAlignTableAxisY2.commands.saveConfiguration := FALSE;
   cmAnodeAlignTableAxisY2.commands.uploadCurrentTorque := FALSE;
   cmAnodeAlignTableAxisY2.commands.reset := FALSE;
   cmAnodeAlignTableAxisY2.monitoring.enable := TRUE;
   cmAnodeAlignTableAxisY2.monitoring.referenceDesignator := WSTRING#'AnodeAlignTableAxisY2';
   cmAnodeAlignTableAxisY2.monitoring.enabled := TRUE;
   cmAnodeAlignTableAxisY2.monitoring.enableManualCmds := FALSE;
   cmAnodeAlignTableAxisY2.monitoring.reset := FALSE;
   cmAnodeAlignTableAxisY2.monitoring.resetAxis := FALSE;
   cmAnodeAlignTableAxisY2.monitoring.enableAxis := TRUE;
   cmAnodeAlignTableAxisY2.monitoring.openBrake := FALSE;
   cmAnodeAlignTableAxisY2.monitoring.jogBackward := FALSE;
   cmAnodeAlignTableAxisY2.monitoring.jogForward := FALSE;
   cmAnodeAlignTableAxisY2.monitoring.moveVelocity := FALSE;
   cmAnodeAlignTableAxisY2.monitoring.stop := FALSE;
   cmAnodeAlignTableAxisY2.monitoring.fastStop := FALSE;
   cmAnodeAlignTableAxisY2.monitoring.torqueLimiting := FALSE;
   cmAnodeAlignTableAxisY2.monitoring.homing := FALSE;
   cmAnodeAlignTableAxisY2.monitoring.posRelative := FALSE;
   cmAnodeAlignTableAxisY2.monitoring.posAbsolute := FALSE;
   cmAnodeAlignTableAxisY2.monitoring.posSuperimposed := FALSE;
   cmAnodeAlignTableAxisY2.monitoring.haltSuperimposed := FALSE;
   cmAnodeAlignTableAxisY2.monitoring.brakeOpened := FALSE;
   cmAnodeAlignTableAxisY2.monitoring.axisEnabled := TRUE;
   cmAnodeAlignTableAxisY2.monitoring.resetActive := FALSE;
   cmAnodeAlignTableAxisY2.monitoring.inVelocity := FALSE;
   cmAnodeAlignTableAxisY2.monitoring.inLimitation := FALSE;
   cmAnodeAlignTableAxisY2.monitoring.inClamping := FALSE;
   cmAnodeAlignTableAxisY2.monitoring.startSync := FALSE;
   cmAnodeAlignTableAxisY2.monitoring.inSync := FALSE;
   cmAnodeAlignTableAxisY2.monitoring.inSimulation := FALSE;
   cmAnodeAlignTableAxisY2.monitoring.jogSelected := FALSE;
   cmAnodeAlignTableAxisY2.monitoring.moveVelocitySelected := FALSE;
   cmAnodeAlignTableAxisY2.monitoring.stopSelected := FALSE;
   cmAnodeAlignTableAxisY2.monitoring.fastStopSelected := FALSE;
   cmAnodeAlignTableAxisY2.monitoring.torqueLimitingSelected := FALSE;
   cmAnodeAlignTableAxisY2.monitoring.homingSelected := FALSE;
   cmAnodeAlignTableAxisY2.monitoring.posRelativeSelected := FALSE;
   cmAnodeAlignTableAxisY2.monitoring.posAbsoluteSelected := FALSE;
   cmAnodeAlignTableAxisY2.monitoring.posSuperimposedSelected := FALSE;
   cmAnodeAlignTableAxisY2.monitoring.haltSuperimposedSelected := FALSE;
   cmAnodeAlignTableAxisY2.monitoring.commandBusy := FALSE;
   cmAnodeAlignTableAxisY2.monitoring.commandDone := FALSE;
   cmAnodeAlignTableAxisY2.monitoring.commandAborted := FALSE;
   cmAnodeAlignTableAxisY2.monitoring.homingCommandBusy := FALSE;
   cmAnodeAlignTableAxisY2.monitoring.homingCommandDone := FALSE;
   cmAnodeAlignTableAxisY2.monitoring.homingCommandAborted := FALSE;
   cmAnodeAlignTableAxisY2.monitoring.superimposedBusy := FALSE;
   cmAnodeAlignTableAxisY2.monitoring.superimposedDone := FALSE;
   cmAnodeAlignTableAxisY2.monitoring.superimposedAborted := FALSE;
   cmAnodeAlignTableAxisY2.monitoring.selectSetPosition := -1;
   cmAnodeAlignTableAxisY2.monitoring.selectionController := FALSE;
   cmAnodeAlignTableAxisY2.monitoring.interlockGeneral := TRUE;
   cmAnodeAlignTableAxisY2.monitoring.interlockJogForward := TRUE;
   cmAnodeAlignTableAxisY2.monitoring.interlockJogBackward := TRUE;
   cmAnodeAlignTableAxisY2.monitoring.interlockWarningGeneral := FALSE;
   cmAnodeAlignTableAxisY2.monitoring.interlockWarningJogForward := FALSE;
   cmAnodeAlignTableAxisY2.monitoring.interlockWarningJogBackward := FALSE;
   cmAnodeAlignTableAxisY2.monitoring.valid := TRUE;
   cmAnodeAlignTableAxisY2.monitoring.busy := TRUE;
   cmAnodeAlignTableAxisY2.monitoring.error := FALSE;
   cmAnodeAlignTableAxisY2.monitoring.status := 16#7002;
   cmAnodeAlignTableAxisY2.monitoring.subfunctionStatus := 16#0000;
   cmAnodeAlignTableAxisY2.monitoring.actualPosition := 0.0;
   cmAnodeAlignTableAxisY2.monitoring.actualSpeed := 0.0;
   cmAnodeAlignTableAxisY2.monitoring.speedUnit := 1062;
   cmAnodeAlignTableAxisY2.monitoring.positionUnit := 1013;
   cmAnodeAlignTableAxisY2.monitoring.axisStatus1 := 16#0200_10E1;
   cmAnodeAlignTableAxisY2.monitoring.axisStatus2 := 16#0000_0000;
   cmAnodeAlignTableAxisY2.monitoring.axisType := 1;
   cmAnodeAlignTableAxisY2.monitoring.maxVelocity := 2500.0;
   cmAnodeAlignTableAxisY2.monitoring.actualCurrent := 0.0;
   cmAnodeAlignTableAxisY2.monitoring.actualTorque := 0.0;
   cmAnodeAlignTableAxisY2.monitoring.velocityOverrideEnabled := FALSE;
   cmAnodeAlignTableAxisY2.monitoring.sinaParaError := FALSE;
   cmAnodeAlignTableAxisY2.monitoring.sinaParaStatus := 16#0000_0000;
   cmAnodeAlignTableAxisY2.configuration.referenceDesignator := WSTRING#'AnodeAlignTableAxisY2';
   cmAnodeAlignTableAxisY2.configuration.disableAlarms := FALSE;
   cmAnodeAlignTableAxisY2.configuration.masterControlPopUp := TRUE;
   cmAnodeAlignTableAxisY2.configuration.setPositions[0].position := 0.0;
   cmAnodeAlignTableAxisY2.configuration.setPositions[1].position := 3.0;
   cmAnodeAlignTableAxisY2.configuration.setPositions[2..9].position := 0.0;
   cmAnodeAlignTableAxisY2.configuration.setPositions[10].position := 8.5;
   cmAnodeAlignTableAxisY2.configuration.setPositions[11..15].position := 0.0;
   cmAnodeAlignTableAxisY2.configuration.setPositions[0..1].velocity := 50.0;
   cmAnodeAlignTableAxisY2.configuration.setPositions[2..15].velocity := -1.0;
   cmAnodeAlignTableAxisY2.configuration.setPositions[0..1].acceleration := 500.0;
   cmAnodeAlignTableAxisY2.configuration.setPositions[2..15].acceleration := -1.0;
   cmAnodeAlignTableAxisY2.configuration.setPositions[0..1].deceleration := 500.0;
   cmAnodeAlignTableAxisY2.configuration.setPositions[2..15].deceleration := -1.0;
   cmAnodeAlignTableAxisY2.configuration.setPositions[0..15]."name" := '';
   cmAnodeMainPnP1RotaryCwCcw.commands.refreshConfiguration := FALSE;
   cmAnodeMainPnP1RotaryCwCcw.commands.editConfiguration := FALSE;
   cmAnodeMainPnP1RotaryCwCcw.commands.saveConfiguration := FALSE;
   cmAnodeMainPnP1RotaryCwCcw.commands.reset := FALSE;
   cmAnodeMainPnP1RotaryCwCcw.commands.commandHomePos := FALSE;
   cmAnodeMainPnP1RotaryCwCcw.commands.commandWorkPos := FALSE;
   cmAnodeMainPnP1RotaryCwCcw.monitoring.enable := TRUE;
   cmAnodeMainPnP1RotaryCwCcw.monitoring.referenceDesignator := WSTRING#'MainPnP1RotaryCwCcw';
   cmAnodeMainPnP1RotaryCwCcw.monitoring.commandHomePos := FALSE;
   cmAnodeMainPnP1RotaryCwCcw.monitoring.commandWorkPos := FALSE;
   cmAnodeMainPnP1RotaryCwCcw.monitoring.goToHomePos := FALSE;
   cmAnodeMainPnP1RotaryCwCcw.monitoring.goToWorkPos := TRUE;
   cmAnodeMainPnP1RotaryCwCcw.monitoring.inHomePos := FALSE;
   cmAnodeMainPnP1RotaryCwCcw.monitoring.inWorkPos := TRUE;
   cmAnodeMainPnP1RotaryCwCcw.monitoring.reset := FALSE;
   cmAnodeMainPnP1RotaryCwCcw.monitoring.enableManualCmds := FALSE;
   cmAnodeMainPnP1RotaryCwCcw.monitoring.error := FALSE;
   cmAnodeMainPnP1RotaryCwCcw.monitoring.interlockHomePos := TRUE;
   cmAnodeMainPnP1RotaryCwCcw.monitoring.interlockWorkPos := TRUE;
   cmAnodeMainPnP1RotaryCwCcw.monitoring.status := 16#7006;
   cmAnodeMainPnP1RotaryCwCcw.monitoring.interlockWarningWorkPos := FALSE;
   cmAnodeMainPnP1RotaryCwCcw.monitoring.interlockWarningHomePos := FALSE;
   cmAnodeMainPnP1RotaryCwCcw.configuration.referenceDesignator := WSTRING#'MainPnP1RotaryCwCcw';
   cmAnodeMainPnP1RotaryCwCcw.configuration.monitoringLeavingFeedback := T#5S;
   cmAnodeMainPnP1RotaryCwCcw.configuration.monitoringReachingFeedback := T#5S;
   cmAnodeMainPnP1RotaryCwCcw.configuration.monitoringDiscrepancy := T#0MS;
   cmAnodeMainPnP1RotaryCwCcw.configuration.setOutputHomeContinuously := TRUE;
   cmAnodeMainPnP1RotaryCwCcw.configuration.setOutputWorkContinuously := TRUE;
   cmAnodeMainPnP1RotaryCwCcw.configuration.disableHomeCommand := FALSE;
   cmAnodeMainPnP1RotaryCwCcw.configuration.disableFeedbackHomePos := TRUE;
   cmAnodeMainPnP1RotaryCwCcw.configuration.disableFeedbackWorkPos := TRUE;
   cmAnodeMainPnP1RotaryCwCcw.configuration.disableAlarms := TRUE;
   cmAnodeMainPnP1RotaryCwCcw.configuration.resetOutputsOnError := FALSE;
   cmAnodeMainPnP1RotaryCwCcw.configuration.allwaysWaitOnReachingTime := FALSE;
   cmAnodeMainPnP1SuctionPlateVacuum.commands.refreshConfiguration := FALSE;
   cmAnodeMainPnP1SuctionPlateVacuum.commands.editConfiguration := FALSE;
   cmAnodeMainPnP1SuctionPlateVacuum.commands.saveConfiguration := FALSE;
   cmAnodeMainPnP1SuctionPlateVacuum.commands.reset := FALSE;
   cmAnodeMainPnP1SuctionPlateVacuum.commands.commandHomePos := FALSE;
   cmAnodeMainPnP1SuctionPlateVacuum.commands.commandWorkPos := FALSE;
   cmAnodeMainPnP1SuctionPlateVacuum.monitoring.enable := TRUE;
   cmAnodeMainPnP1SuctionPlateVacuum.monitoring.referenceDesignator := WSTRING#'MainPnP1Vacuum';
   cmAnodeMainPnP1SuctionPlateVacuum.monitoring.commandHomePos := TRUE;
   cmAnodeMainPnP1SuctionPlateVacuum.monitoring.commandWorkPos := FALSE;
   cmAnodeMainPnP1SuctionPlateVacuum.monitoring.goToHomePos := TRUE;
   cmAnodeMainPnP1SuctionPlateVacuum.monitoring.goToWorkPos := FALSE;
   cmAnodeMainPnP1SuctionPlateVacuum.monitoring.inHomePos := TRUE;
   cmAnodeMainPnP1SuctionPlateVacuum.monitoring.inWorkPos := FALSE;
   cmAnodeMainPnP1SuctionPlateVacuum.monitoring.reset := FALSE;
   cmAnodeMainPnP1SuctionPlateVacuum.monitoring.enableManualCmds := FALSE;
   cmAnodeMainPnP1SuctionPlateVacuum.monitoring.error := FALSE;
   cmAnodeMainPnP1SuctionPlateVacuum.monitoring.interlockHomePos := TRUE;
   cmAnodeMainPnP1SuctionPlateVacuum.monitoring.interlockWorkPos := TRUE;
   cmAnodeMainPnP1SuctionPlateVacuum.monitoring.status := 16#7004;
   cmAnodeMainPnP1SuctionPlateVacuum.monitoring.interlockWarningWorkPos := FALSE;
   cmAnodeMainPnP1SuctionPlateVacuum.monitoring.interlockWarningHomePos := FALSE;
   cmAnodeMainPnP1SuctionPlateVacuum.configuration.referenceDesignator := WSTRING#'MainPnP1Vacuum';
   cmAnodeMainPnP1SuctionPlateVacuum.configuration.monitoringLeavingFeedback := T#100MS;
   cmAnodeMainPnP1SuctionPlateVacuum.configuration.monitoringReachingFeedback := T#100MS;
   cmAnodeMainPnP1SuctionPlateVacuum.configuration.monitoringDiscrepancy := T#15S;
   cmAnodeMainPnP1SuctionPlateVacuum.configuration.setOutputHomeContinuously := TRUE;
   cmAnodeMainPnP1SuctionPlateVacuum.configuration.setOutputWorkContinuously := TRUE;
   cmAnodeMainPnP1SuctionPlateVacuum.configuration.disableHomeCommand := FALSE;
   cmAnodeMainPnP1SuctionPlateVacuum.configuration.disableFeedbackHomePos := FALSE;
   cmAnodeMainPnP1SuctionPlateVacuum.configuration.disableFeedbackWorkPos := FALSE;
   cmAnodeMainPnP1SuctionPlateVacuum.configuration.disableAlarms := FALSE;
   cmAnodeMainPnP1SuctionPlateVacuum.configuration.resetOutputsOnError := FALSE;
   cmAnodeMainPnP1SuctionPlateVacuum.configuration.allwaysWaitOnReachingTime := FALSE;
   cmAnodeMainPnP2SuctionPlateVacuum.commands.refreshConfiguration := FALSE;
   cmAnodeMainPnP2SuctionPlateVacuum.commands.editConfiguration := FALSE;
   cmAnodeMainPnP2SuctionPlateVacuum.commands.saveConfiguration := FALSE;
   cmAnodeMainPnP2SuctionPlateVacuum.commands.reset := FALSE;
   cmAnodeMainPnP2SuctionPlateVacuum.commands.commandHomePos := FALSE;
   cmAnodeMainPnP2SuctionPlateVacuum.commands.commandWorkPos := FALSE;
   cmAnodeMainPnP2SuctionPlateVacuum.monitoring.enable := TRUE;
   cmAnodeMainPnP2SuctionPlateVacuum.monitoring.referenceDesignator := WSTRING#'MainPnP2Vacuum';
   cmAnodeMainPnP2SuctionPlateVacuum.monitoring.commandHomePos := TRUE;
   cmAnodeMainPnP2SuctionPlateVacuum.monitoring.commandWorkPos := FALSE;
   cmAnodeMainPnP2SuctionPlateVacuum.monitoring.goToHomePos := TRUE;
   cmAnodeMainPnP2SuctionPlateVacuum.monitoring.goToWorkPos := FALSE;
   cmAnodeMainPnP2SuctionPlateVacuum.monitoring.inHomePos := TRUE;
   cmAnodeMainPnP2SuctionPlateVacuum.monitoring.inWorkPos := FALSE;
   cmAnodeMainPnP2SuctionPlateVacuum.monitoring.reset := FALSE;
   cmAnodeMainPnP2SuctionPlateVacuum.monitoring.enableManualCmds := FALSE;
   cmAnodeMainPnP2SuctionPlateVacuum.monitoring.error := FALSE;
   cmAnodeMainPnP2SuctionPlateVacuum.monitoring.interlockHomePos := TRUE;
   cmAnodeMainPnP2SuctionPlateVacuum.monitoring.interlockWorkPos := TRUE;
   cmAnodeMainPnP2SuctionPlateVacuum.monitoring.status := 16#7004;
   cmAnodeMainPnP2SuctionPlateVacuum.monitoring.interlockWarningWorkPos := FALSE;
   cmAnodeMainPnP2SuctionPlateVacuum.monitoring.interlockWarningHomePos := FALSE;
   cmAnodeMainPnP2SuctionPlateVacuum.configuration.referenceDesignator := WSTRING#'MainPnP2Vacuum';
   cmAnodeMainPnP2SuctionPlateVacuum.configuration.monitoringLeavingFeedback := T#100MS;
   cmAnodeMainPnP2SuctionPlateVacuum.configuration.monitoringReachingFeedback := T#100MS;
   cmAnodeMainPnP2SuctionPlateVacuum.configuration.monitoringDiscrepancy := T#15S;
   cmAnodeMainPnP2SuctionPlateVacuum.configuration.setOutputHomeContinuously := TRUE;
   cmAnodeMainPnP2SuctionPlateVacuum.configuration.setOutputWorkContinuously := TRUE;
   cmAnodeMainPnP2SuctionPlateVacuum.configuration.disableHomeCommand := FALSE;
   cmAnodeMainPnP2SuctionPlateVacuum.configuration.disableFeedbackHomePos := FALSE;
   cmAnodeMainPnP2SuctionPlateVacuum.configuration.disableFeedbackWorkPos := FALSE;
   cmAnodeMainPnP2SuctionPlateVacuum.configuration.disableAlarms := FALSE;
   cmAnodeMainPnP2SuctionPlateVacuum.configuration.resetOutputsOnError := FALSE;
   cmAnodeMainPnP2SuctionPlateVacuum.configuration.allwaysWaitOnReachingTime := FALSE;
   cmAnodeAlignTableSuctionPlateVacuum.commands.refreshConfiguration := FALSE;
   cmAnodeAlignTableSuctionPlateVacuum.commands.editConfiguration := FALSE;
   cmAnodeAlignTableSuctionPlateVacuum.commands.saveConfiguration := FALSE;
   cmAnodeAlignTableSuctionPlateVacuum.commands.reset := FALSE;
   cmAnodeAlignTableSuctionPlateVacuum.commands.commandHomePos := FALSE;
   cmAnodeAlignTableSuctionPlateVacuum.commands.commandWorkPos := FALSE;
   cmAnodeAlignTableSuctionPlateVacuum.monitoring.enable := TRUE;
   cmAnodeAlignTableSuctionPlateVacuum.monitoring.referenceDesignator := WSTRING#'AlignTableVaccum';
   cmAnodeAlignTableSuctionPlateVacuum.monitoring.commandHomePos := TRUE;
   cmAnodeAlignTableSuctionPlateVacuum.monitoring.commandWorkPos := FALSE;
   cmAnodeAlignTableSuctionPlateVacuum.monitoring.goToHomePos := TRUE;
   cmAnodeAlignTableSuctionPlateVacuum.monitoring.goToWorkPos := FALSE;
   cmAnodeAlignTableSuctionPlateVacuum.monitoring.inHomePos := TRUE;
   cmAnodeAlignTableSuctionPlateVacuum.monitoring.inWorkPos := FALSE;
   cmAnodeAlignTableSuctionPlateVacuum.monitoring.reset := FALSE;
   cmAnodeAlignTableSuctionPlateVacuum.monitoring.enableManualCmds := FALSE;
   cmAnodeAlignTableSuctionPlateVacuum.monitoring.error := FALSE;
   cmAnodeAlignTableSuctionPlateVacuum.monitoring.interlockHomePos := TRUE;
   cmAnodeAlignTableSuctionPlateVacuum.monitoring.interlockWorkPos := TRUE;
   cmAnodeAlignTableSuctionPlateVacuum.monitoring.status := 16#7004;
   cmAnodeAlignTableSuctionPlateVacuum.monitoring.interlockWarningWorkPos := FALSE;
   cmAnodeAlignTableSuctionPlateVacuum.monitoring.interlockWarningHomePos := FALSE;
   cmAnodeAlignTableSuctionPlateVacuum.configuration.referenceDesignator := WSTRING#'AlignTableVaccum';
   cmAnodeAlignTableSuctionPlateVacuum.configuration.monitoringLeavingFeedback := T#3S;
   cmAnodeAlignTableSuctionPlateVacuum.configuration.monitoringReachingFeedback := T#3S;
   cmAnodeAlignTableSuctionPlateVacuum.configuration.monitoringDiscrepancy := T#15MS;
   cmAnodeAlignTableSuctionPlateVacuum.configuration.setOutputHomeContinuously := TRUE;
   cmAnodeAlignTableSuctionPlateVacuum.configuration.setOutputWorkContinuously := TRUE;
   cmAnodeAlignTableSuctionPlateVacuum.configuration.disableHomeCommand := FALSE;
   cmAnodeAlignTableSuctionPlateVacuum.configuration.disableFeedbackHomePos := FALSE;
   cmAnodeAlignTableSuctionPlateVacuum.configuration.disableFeedbackWorkPos := FALSE;
   cmAnodeAlignTableSuctionPlateVacuum.configuration.disableAlarms := FALSE;
   cmAnodeAlignTableSuctionPlateVacuum.configuration.resetOutputsOnError := FALSE;
   cmAnodeAlignTableSuctionPlateVacuum.configuration.allwaysWaitOnReachingTime := FALSE;
   cmAnodeGlassCleaning.commands.refreshConfiguration := FALSE;
   cmAnodeGlassCleaning.commands.editConfiguration := FALSE;
   cmAnodeGlassCleaning.commands.saveConfiguration := FALSE;
   cmAnodeGlassCleaning.commands.reset := FALSE;
   cmAnodeGlassCleaning.commands.commandHomePos := FALSE;
   cmAnodeGlassCleaning.commands.commandWorkPos := FALSE;
   cmAnodeGlassCleaning.monitoring.enable := TRUE;
   cmAnodeGlassCleaning.monitoring.referenceDesignator := WSTRING#'GlassCleaning';
   cmAnodeGlassCleaning.monitoring.commandHomePos := FALSE;
   cmAnodeGlassCleaning.monitoring.commandWorkPos := FALSE;
   cmAnodeGlassCleaning.monitoring.goToHomePos := FALSE;
   cmAnodeGlassCleaning.monitoring.goToWorkPos := TRUE;
   cmAnodeGlassCleaning.monitoring.inHomePos := FALSE;
   cmAnodeGlassCleaning.monitoring.inWorkPos := TRUE;
   cmAnodeGlassCleaning.monitoring.reset := FALSE;
   cmAnodeGlassCleaning.monitoring.enableManualCmds := FALSE;
   cmAnodeGlassCleaning.monitoring.error := FALSE;
   cmAnodeGlassCleaning.monitoring.interlockHomePos := TRUE;
   cmAnodeGlassCleaning.monitoring.interlockWorkPos := TRUE;
   cmAnodeGlassCleaning.monitoring.status := 16#7006;
   cmAnodeGlassCleaning.monitoring.interlockWarningWorkPos := FALSE;
   cmAnodeGlassCleaning.monitoring.interlockWarningHomePos := FALSE;
   cmAnodeGlassCleaning.configuration.referenceDesignator := WSTRING#'GlassCleaning';
   cmAnodeGlassCleaning.configuration.monitoringLeavingFeedback := T#5S;
   cmAnodeGlassCleaning.configuration.monitoringReachingFeedback := T#5S;
   cmAnodeGlassCleaning.configuration.monitoringDiscrepancy := T#0MS;
   cmAnodeGlassCleaning.configuration.setOutputHomeContinuously := TRUE;
   cmAnodeGlassCleaning.configuration.setOutputWorkContinuously := TRUE;
   cmAnodeGlassCleaning.configuration.disableHomeCommand := FALSE;
   cmAnodeGlassCleaning.configuration.disableFeedbackHomePos := TRUE;
   cmAnodeGlassCleaning.configuration.disableFeedbackWorkPos := TRUE;
   cmAnodeGlassCleaning.configuration.disableAlarms := FALSE;
   cmAnodeGlassCleaning.configuration.resetOutputsOnError := FALSE;
   cmAnodeGlassCleaning.configuration.allwaysWaitOnReachingTime := FALSE;
   cmAnodeNgPnpUpDown.commands.refreshConfiguration := FALSE;
   cmAnodeNgPnpUpDown.commands.editConfiguration := FALSE;
   cmAnodeNgPnpUpDown.commands.saveConfiguration := FALSE;
   cmAnodeNgPnpUpDown.commands.reset := FALSE;
   cmAnodeNgPnpUpDown.commands.commandHomePos := FALSE;
   cmAnodeNgPnpUpDown.commands.commandWorkPos := FALSE;
   cmAnodeNgPnpUpDown.monitoring.enable := TRUE;
   cmAnodeNgPnpUpDown.monitoring.referenceDesignator := WSTRING#'NgPnpUpDown';
   cmAnodeNgPnpUpDown.monitoring.commandHomePos := FALSE;
   cmAnodeNgPnpUpDown.monitoring.commandWorkPos := FALSE;
   cmAnodeNgPnpUpDown.monitoring.goToHomePos := TRUE;
   cmAnodeNgPnpUpDown.monitoring.goToWorkPos := FALSE;
   cmAnodeNgPnpUpDown.monitoring.inHomePos := TRUE;
   cmAnodeNgPnpUpDown.monitoring.inWorkPos := FALSE;
   cmAnodeNgPnpUpDown.monitoring.reset := FALSE;
   cmAnodeNgPnpUpDown.monitoring.enableManualCmds := FALSE;
   cmAnodeNgPnpUpDown.monitoring.error := FALSE;
   cmAnodeNgPnpUpDown.monitoring.interlockHomePos := TRUE;
   cmAnodeNgPnpUpDown.monitoring.interlockWorkPos := TRUE;
   cmAnodeNgPnpUpDown.monitoring.status := 16#7004;
   cmAnodeNgPnpUpDown.monitoring.interlockWarningWorkPos := FALSE;
   cmAnodeNgPnpUpDown.monitoring.interlockWarningHomePos := FALSE;
   cmAnodeNgPnpUpDown.configuration.referenceDesignator := WSTRING#'NgPnpUpDown';
   cmAnodeNgPnpUpDown.configuration.monitoringLeavingFeedback := T#5S;
   cmAnodeNgPnpUpDown.configuration.monitoringReachingFeedback := T#5S;
   cmAnodeNgPnpUpDown.configuration.monitoringDiscrepancy := T#0MS;
   cmAnodeNgPnpUpDown.configuration.setOutputHomeContinuously := TRUE;
   cmAnodeNgPnpUpDown.configuration.setOutputWorkContinuously := TRUE;
   cmAnodeNgPnpUpDown.configuration.disableHomeCommand := FALSE;
   cmAnodeNgPnpUpDown.configuration.disableFeedbackHomePos := TRUE;
   cmAnodeNgPnpUpDown.configuration.disableFeedbackWorkPos := TRUE;
   cmAnodeNgPnpUpDown.configuration.disableAlarms := FALSE;
   cmAnodeNgPnpUpDown.configuration.resetOutputsOnError := FALSE;
   cmAnodeNgPnpUpDown.configuration.allwaysWaitOnReachingTime := FALSE;
   cmAnodeNgPnp1stFwdBwd.commands.refreshConfiguration := FALSE;
   cmAnodeNgPnp1stFwdBwd.commands.editConfiguration := FALSE;
   cmAnodeNgPnp1stFwdBwd.commands.saveConfiguration := FALSE;
   cmAnodeNgPnp1stFwdBwd.commands.reset := FALSE;
   cmAnodeNgPnp1stFwdBwd.commands.commandHomePos := FALSE;
   cmAnodeNgPnp1stFwdBwd.commands.commandWorkPos := FALSE;
   cmAnodeNgPnp1stFwdBwd.monitoring.enable := TRUE;
   cmAnodeNgPnp1stFwdBwd.monitoring.referenceDesignator := WSTRING#'NgPnp1stFwdBwd';
   cmAnodeNgPnp1stFwdBwd.monitoring.commandHomePos := FALSE;
   cmAnodeNgPnp1stFwdBwd.monitoring.commandWorkPos := FALSE;
   cmAnodeNgPnp1stFwdBwd.monitoring.goToHomePos := TRUE;
   cmAnodeNgPnp1stFwdBwd.monitoring.goToWorkPos := FALSE;
   cmAnodeNgPnp1stFwdBwd.monitoring.inHomePos := TRUE;
   cmAnodeNgPnp1stFwdBwd.monitoring.inWorkPos := FALSE;
   cmAnodeNgPnp1stFwdBwd.monitoring.reset := FALSE;
   cmAnodeNgPnp1stFwdBwd.monitoring.enableManualCmds := FALSE;
   cmAnodeNgPnp1stFwdBwd.monitoring.error := FALSE;
   cmAnodeNgPnp1stFwdBwd.monitoring.interlockHomePos := TRUE;
   cmAnodeNgPnp1stFwdBwd.monitoring.interlockWorkPos := TRUE;
   cmAnodeNgPnp1stFwdBwd.monitoring.status := 16#7004;
   cmAnodeNgPnp1stFwdBwd.monitoring.interlockWarningWorkPos := FALSE;
   cmAnodeNgPnp1stFwdBwd.monitoring.interlockWarningHomePos := FALSE;
   cmAnodeNgPnp1stFwdBwd.configuration.referenceDesignator := WSTRING#'TwoWayAct.';
   cmAnodeNgPnp1stFwdBwd.configuration.monitoringLeavingFeedback := T#5S;
   cmAnodeNgPnp1stFwdBwd.configuration.monitoringReachingFeedback := T#5S;
   cmAnodeNgPnp1stFwdBwd.configuration.monitoringDiscrepancy := T#0MS;
   cmAnodeNgPnp1stFwdBwd.configuration.setOutputHomeContinuously := TRUE;
   cmAnodeNgPnp1stFwdBwd.configuration.setOutputWorkContinuously := TRUE;
   cmAnodeNgPnp1stFwdBwd.configuration.disableHomeCommand := FALSE;
   cmAnodeNgPnp1stFwdBwd.configuration.disableFeedbackHomePos := FALSE;
   cmAnodeNgPnp1stFwdBwd.configuration.disableFeedbackWorkPos := FALSE;
   cmAnodeNgPnp1stFwdBwd.configuration.disableAlarms := FALSE;
   cmAnodeNgPnp1stFwdBwd.configuration.resetOutputsOnError := FALSE;
   cmAnodeNgPnp1stFwdBwd.configuration.allwaysWaitOnReachingTime := FALSE;
   cmAnodeNgPnp2ndFwdBwd.commands.refreshConfiguration := FALSE;
   cmAnodeNgPnp2ndFwdBwd.commands.editConfiguration := FALSE;
   cmAnodeNgPnp2ndFwdBwd.commands.saveConfiguration := FALSE;
   cmAnodeNgPnp2ndFwdBwd.commands.reset := FALSE;
   cmAnodeNgPnp2ndFwdBwd.commands.commandHomePos := FALSE;
   cmAnodeNgPnp2ndFwdBwd.commands.commandWorkPos := FALSE;
   cmAnodeNgPnp2ndFwdBwd.monitoring.enable := TRUE;
   cmAnodeNgPnp2ndFwdBwd.monitoring.referenceDesignator := WSTRING#'NgPnp2ndFwdBwd';
   cmAnodeNgPnp2ndFwdBwd.monitoring.commandHomePos := FALSE;
   cmAnodeNgPnp2ndFwdBwd.monitoring.commandWorkPos := FALSE;
   cmAnodeNgPnp2ndFwdBwd.monitoring.goToHomePos := FALSE;
   cmAnodeNgPnp2ndFwdBwd.monitoring.goToWorkPos := FALSE;
   cmAnodeNgPnp2ndFwdBwd.monitoring.inHomePos := TRUE;
   cmAnodeNgPnp2ndFwdBwd.monitoring.inWorkPos := FALSE;
   cmAnodeNgPnp2ndFwdBwd.monitoring.reset := FALSE;
   cmAnodeNgPnp2ndFwdBwd.monitoring.enableManualCmds := FALSE;
   cmAnodeNgPnp2ndFwdBwd.monitoring.error := FALSE;
   cmAnodeNgPnp2ndFwdBwd.monitoring.interlockHomePos := TRUE;
   cmAnodeNgPnp2ndFwdBwd.monitoring.interlockWorkPos := TRUE;
   cmAnodeNgPnp2ndFwdBwd.monitoring.status := 16#7004;
   cmAnodeNgPnp2ndFwdBwd.monitoring.interlockWarningWorkPos := FALSE;
   cmAnodeNgPnp2ndFwdBwd.monitoring.interlockWarningHomePos := FALSE;
   cmAnodeNgPnp2ndFwdBwd.configuration.referenceDesignator := WSTRING#'TwoWayAct.';
   cmAnodeNgPnp2ndFwdBwd.configuration.monitoringLeavingFeedback := T#5S;
   cmAnodeNgPnp2ndFwdBwd.configuration.monitoringReachingFeedback := T#5S;
   cmAnodeNgPnp2ndFwdBwd.configuration.monitoringDiscrepancy := T#0MS;
   cmAnodeNgPnp2ndFwdBwd.configuration.setOutputHomeContinuously := TRUE;
   cmAnodeNgPnp2ndFwdBwd.configuration.setOutputWorkContinuously := TRUE;
   cmAnodeNgPnp2ndFwdBwd.configuration.disableHomeCommand := FALSE;
   cmAnodeNgPnp2ndFwdBwd.configuration.disableFeedbackHomePos := FALSE;
   cmAnodeNgPnp2ndFwdBwd.configuration.disableFeedbackWorkPos := FALSE;
   cmAnodeNgPnp2ndFwdBwd.configuration.disableAlarms := FALSE;
   cmAnodeNgPnp2ndFwdBwd.configuration.resetOutputsOnError := FALSE;
   cmAnodeNgPnp2ndFwdBwd.configuration.allwaysWaitOnReachingTime := FALSE;
   cmAnodeMaintenanceMovingFixFrontRearFwdBwd.commands.refreshConfiguration := FALSE;
   cmAnodeMaintenanceMovingFixFrontRearFwdBwd.commands.editConfiguration := FALSE;
   cmAnodeMaintenanceMovingFixFrontRearFwdBwd.commands.saveConfiguration := FALSE;
   cmAnodeMaintenanceMovingFixFrontRearFwdBwd.commands.reset := FALSE;
   cmAnodeMaintenanceMovingFixFrontRearFwdBwd.commands.commandHomePos := FALSE;
   cmAnodeMaintenanceMovingFixFrontRearFwdBwd.commands.commandWorkPos := FALSE;
   cmAnodeMaintenanceMovingFixFrontRearFwdBwd.monitoring.enable := TRUE;
   cmAnodeMaintenanceMovingFixFrontRearFwdBwd.monitoring.referenceDesignator := WSTRING#'MaintenanceFix';
   cmAnodeMaintenanceMovingFixFrontRearFwdBwd.monitoring.commandHomePos := FALSE;
   cmAnodeMaintenanceMovingFixFrontRearFwdBwd.monitoring.commandWorkPos := FALSE;
   cmAnodeMaintenanceMovingFixFrontRearFwdBwd.monitoring.goToHomePos := FALSE;
   cmAnodeMaintenanceMovingFixFrontRearFwdBwd.monitoring.goToWorkPos := FALSE;
   cmAnodeMaintenanceMovingFixFrontRearFwdBwd.monitoring.inHomePos := FALSE;
   cmAnodeMaintenanceMovingFixFrontRearFwdBwd.monitoring.inWorkPos := FALSE;
   cmAnodeMaintenanceMovingFixFrontRearFwdBwd.monitoring.reset := FALSE;
   cmAnodeMaintenanceMovingFixFrontRearFwdBwd.monitoring.enableManualCmds := FALSE;
   cmAnodeMaintenanceMovingFixFrontRearFwdBwd.monitoring.error := FALSE;
   cmAnodeMaintenanceMovingFixFrontRearFwdBwd.monitoring.interlockHomePos := TRUE;
   cmAnodeMaintenanceMovingFixFrontRearFwdBwd.monitoring.interlockWorkPos := TRUE;
   cmAnodeMaintenanceMovingFixFrontRearFwdBwd.monitoring.status := 16#7003;
   cmAnodeMaintenanceMovingFixFrontRearFwdBwd.monitoring.interlockWarningWorkPos := FALSE;
   cmAnodeMaintenanceMovingFixFrontRearFwdBwd.monitoring.interlockWarningHomePos := FALSE;
   cmAnodeMaintenanceMovingFixFrontRearFwdBwd.configuration.referenceDesignator := WSTRING#'TwoWayAct.';
   cmAnodeMaintenanceMovingFixFrontRearFwdBwd.configuration.monitoringLeavingFeedback := T#5S;
   cmAnodeMaintenanceMovingFixFrontRearFwdBwd.configuration.monitoringReachingFeedback := T#5S;
   cmAnodeMaintenanceMovingFixFrontRearFwdBwd.configuration.monitoringDiscrepancy := T#0MS;
   cmAnodeMaintenanceMovingFixFrontRearFwdBwd.configuration.setOutputHomeContinuously := TRUE;
   cmAnodeMaintenanceMovingFixFrontRearFwdBwd.configuration.setOutputWorkContinuously := TRUE;
   cmAnodeMaintenanceMovingFixFrontRearFwdBwd.configuration.disableHomeCommand := FALSE;
   cmAnodeMaintenanceMovingFixFrontRearFwdBwd.configuration.disableFeedbackHomePos := FALSE;
   cmAnodeMaintenanceMovingFixFrontRearFwdBwd.configuration.disableFeedbackWorkPos := FALSE;
   cmAnodeMaintenanceMovingFixFrontRearFwdBwd.configuration.disableAlarms := FALSE;
   cmAnodeMaintenanceMovingFixFrontRearFwdBwd.configuration.resetOutputsOnError := FALSE;
   cmAnodeMaintenanceMovingFixFrontRearFwdBwd.configuration.allwaysWaitOnReachingTime := FALSE;
   cmAnodeNgBoxLiftUpDown.commands.refreshConfiguration := FALSE;
   cmAnodeNgBoxLiftUpDown.commands.editConfiguration := FALSE;
   cmAnodeNgBoxLiftUpDown.commands.saveConfiguration := FALSE;
   cmAnodeNgBoxLiftUpDown.commands.reset := FALSE;
   cmAnodeNgBoxLiftUpDown.commands.commandHomePos := FALSE;
   cmAnodeNgBoxLiftUpDown.commands.commandWorkPos := FALSE;
   cmAnodeNgBoxLiftUpDown.monitoring.enable := TRUE;
   cmAnodeNgBoxLiftUpDown.monitoring.referenceDesignator := WSTRING#'NgBoxLiftUpDown';
   cmAnodeNgBoxLiftUpDown.monitoring.commandHomePos := FALSE;
   cmAnodeNgBoxLiftUpDown.monitoring.commandWorkPos := FALSE;
   cmAnodeNgBoxLiftUpDown.monitoring.goToHomePos := FALSE;
   cmAnodeNgBoxLiftUpDown.monitoring.goToWorkPos := TRUE;
   cmAnodeNgBoxLiftUpDown.monitoring.inHomePos := FALSE;
   cmAnodeNgBoxLiftUpDown.monitoring.inWorkPos := TRUE;
   cmAnodeNgBoxLiftUpDown.monitoring.reset := FALSE;
   cmAnodeNgBoxLiftUpDown.monitoring.enableManualCmds := FALSE;
